(* Logix 5000 project; controller ARS14002_PLC vendor 1 type 14 code 218 rev 30.11; software revision 30.01; part 11 of 13 *)
(* tags used below, declared in another part *)
   AN_1000C : CM_AI_SCL;
   AN_1000C_SP : INT;
   AN_200A : CM_AI_SCL;
   AN_200A_SP : REAL;
   AT2_HIBON_DISCHARGE_TEMP_MAX : REAL;
   AT2_PLANT_ATOMIZING : BOOL;
   AT2_PLANT_ATOMIZING_ONS : BOOL;
   AT2_PLANT_COLLECTING : BOOL;
   AT2_PLANT_COLLECTION_TIME : TIMER;
   AT2_PLANT_GOOD_GAS_TIME : TIMER;   // AT2 total time with good gas and no collection stops
   AT2_PLANT_GOOD_H2O_TIME : TIMER;   // AT2 time with good dew point and no collection stop
   AT2_PLANT_GOOD_O2_TIME : TIMER;   // AT2 time with good O2 and no collection stop
   AT2_PLANT_H2O_MIN : REAL;   // AT2 Heat Minimum after burp
   AT2_PLANT_LIKELY_COLLECTING : BOOL;
   AT2_PLANT_LIKELY_COLLECTION_TIME : TIMER;
   AT2_PLANT_MAX_H2O : REAL;
   AT2_PLANT_MAX_O2 : REAL;
   AT2_PLANT_O2_MIN : REAL;   // AT2 Heat Minimum after burp
   AT3_HIBON_DISCHARGE_TEMP_MAX : REAL;
   AT3_PLANT_ATOMIZING : BOOL;
   AT3_PLANT_ATOMIZING_ONS : BOOL;
   AT3_PLANT_COLLECTING : BOOL;
   AT3_PLANT_COLLECTION_TIME : TIMER;
   AT3_PLANT_GOOD_GAS_TIME : TIMER;   // total time with good gas and no collection stops
   AT3_PLANT_GOOD_H2O_TIME : TIMER;   // time with good dew point and no collection stop
   AT3_PLANT_GOOD_O2_TIME : TIMER;   // time with good O2 and no collection stop
   AT3_PLANT_H2O_MIN : REAL;   // AT3 Plant Minimum after burp
   AT3_PLANT_LIKELY_COLLECTING : BOOL;
   AT3_PLANT_LIKELY_COLLECTION_TIME : TIMER;
   AT3_PLANT_MAX_H2O : REAL;
   AT3_PLANT_MAX_O2 : REAL;
   AT3_PLANT_O2_MIN : REAL;   // AT3 Plant Minimum after burp
   CALC_FT_1002_MONTH_RETURN : REAL;
   CALC_FT_1002_MONTH_TOTALIZER_RESET : BOOL;
   CALC_FT_1002_MONTH_TOTALIZER_START : BOOL;
   CALC_FT_1002_MONTH_TOTALIZER_STOP : BOOL;
   Calc_FT_1002_Return_Total : DINT[2100,13];
   Calc_Month : INT;
   CALC_NEXT_DAY_OSR_OB : BOOL;
   CALC_NEXT_DAY_OSR_SB : BOOL;
   CALC_NEXT_MONTH_OSR_OB : BOOL;
   CALC_NEXT_MONTH_OSR_SB : BOOL;
   Calc_TK_700_Fill_Lvl : REAL;
   Calc_TK_700_Fill_Start_Lvl : REAL;
   Calc_TK_700_Fill_Total : DINT[2100,13];
   Calc_TK_700_Month_Fill : REAL;
   Calc_TK_700_Month_Totalizer_Start : BOOL;
   Calc_TK_700_Month_Totalizer_Stop : BOOL;
   Calc_Year : INT;
   Collect_Stop_Dew_Pt : BOOL;
   Collect_Stop_O2 : BOOL;
   COLLECTION_ESTIMATE_SCALING_FACTOR : REAL;
   COLLECTION_LIKELY_PERCENTAGE : REAL;
   Cooldown_Complete_ONS_OB : BOOL;
   Cooldown_Complete_ONS_SB : BOOL;
   COOLDOWN_CYCLES_MIN : DINT[10];
   COOLDOWN_CYCLES_SEC : DINT[10];
   COOLDOWN_TIMER1 : TIMER;
   COOLDOWN_TIMER1_MIN : DINT;
   COOLDOWN_TIMER1_MS : DINT;
   COOLDOWN_TIMER1_SEC : DINT;
   CP_Run : BOOL;
   CP_Run_Atomize : BOOL;
   CP_Run_ONS_OB : BOOL;
   CP_Run_Standby : BOOL;
   CP_RUN_TIMESTAMP_DAY : DINT[10];
   CP_RUN_TIMESTAMP_HOUR : DINT[10];
   CP_RUN_TIMESTAMP_MIN : DINT[10];
   CP_RUN_TIMESTAMP_MONTH : DINT[10];
   CP_RUN_TIMESTAMP_SEC : DINT[10];
   CP_RUN_TIMESTAMP_YEAR : DINT[10];
   FCV_1002 : CM_AO_VLV;
   FCV_101A : CM_AO_VLV;
   FCV_101B : CM_AO_VLV;
   FCV_101C : CM_AO_VLV;
   FCV_102A : CM_AO_VLV;
   FCV_102B : CM_AO_VLV;
   FCV_102C : CM_AO_VLV;
   FCV_202 : CM_AO_VLV;
   FCV_202_COLLECTION_CERTAIN_SP : REAL;
   FCV_202_COLLECTION_LIKELY_SP : REAL;
   FCV_202_OPEN_DLA_TMR : TIMER;
   FCV_204 : CM_AO_VLV;
   FCV_207 : CM_AO_VLV;
   FIT_202_COLLECTION_FLOW : REAL;
   FT_1002 : CM_AI_SCL;
   FT_202 : CM_AI_SCL;
   FVR_800C_EN : BOOL;
   FVR_800D_EN : BOOL;
   HEAT_TIMER_AT2 : TIMER;
   HEAT_TIMER_AT3 : TIMER;
   HEAT_TIMER_PILOT : TIMER;
   P_800A_Cooldown_Complete : BOOL;
   P_800A_Start_Vent_TMR : TIMER;
   P_800B_Cooldown_Complete : BOOL;
   P_800B_Start_Vent_TMR : TIMER;
   P_800C_Cooldown_Complete : BOOL;
   P_800C_Start_Vent_TMR : TIMER;
   P_800D_Cooldown_Complete : BOOL;
   P_800D_Start_Vent_TMR : TIMER;
   PDT_701 : CM_AI_SCL_ALT;
   PIDE_1001 : PID_ENHANCED;
   PIDE_1002 : PID_ENHANCED;
   PIDE_1002_FLOW_SP : PID_ENHANCED;
   PIDE_1221 : PID_ENHANCED;
   PIDE_1251 : PID_ENHANCED;
   PIDE_603 : PID_ENHANCED;
   PIDE_605 : PID_ENHANCED;
   PIDE_753 : PID_ENHANCED;
   PIDE_754 : PID_ENHANCED;
   PIDE_755 : PID_ENHANCED;
   PIDE_800 : PID_ENHANCED;
   PILOT_PLANT_ATOMIZING : BOOL;
   PILOT_PLANT_ATOMIZING_ONS : BOOL;
   PILOT_PLANT_COLLECTING : BOOL;
   PILOT_PLANT_COLLECTION_PERCENT : REAL;
   PILOT_PLANT_COLLECTION_PERCENT_GOOD_GAS : REAL;
   PILOT_PLANT_COLLECTION_TIME : TIMER;
   PILOT_PLANT_GOOD_GAS_PERCENT : REAL;
   PILOT_PLANT_GOOD_GAS_TIME : TIMER;   // PILOT time with good gas and no collection stops
   PILOT_PLANT_GOOD_H2O_PERCENT : REAL;
   PILOT_PLANT_GOOD_H2O_TIME : TIMER;   // PILOT time with good dew point and no collection stop
   PILOT_PLANT_GOOD_O2_PERCENT : REAL;
   PILOT_PLANT_GOOD_O2_TIME : TIMER;   // PILOT time with good O2 and no collection stop
   PILOT_PLANT_H2O_MIN : REAL;   // Pilot Heat Minimum after burp
   PILOT_PLANT_LIKELY_COLLECTING : BOOL;
   PILOT_PLANT_LIKELY_COLLECTION_TIME : TIMER;
   PILOT_PLANT_MAX_H2O : REAL;
   PILOT_PLANT_MAX_O2 : REAL;
   PILOT_PLANT_O2_MIN : REAL;   // Pilot Heat Minimum after burp
   SV_1001F : CM_DO_GENERIC;
   SV_1002F : CM_DO_GENERIC;
   SV_1005X : CM_DO_GENERIC;
   SV_1221F : CM_DO_GENERIC;
   SV_1251F : CM_DO_GENERIC;
   SV_207F : CM_DO_GENERIC;
   SV_603F : CM_DO_GENERIC;
   SV_605F : CM_DO_GENERIC;
   SV_703X : CM_DO_GENERIC;
   SV_753F : CM_DO_GENERIC;
   SV_754F : CM_DO_GENERIC;
   SV_755F : CM_DO_GENERIC;
   TIME_TO_GOOD_GAS_AT2 : REAL;
   TIME_TO_GOOD_GAS_AT3 : REAL;
   TIME_TO_GOOD_GAS_PILOT : REAL;
   TimeStamp : DINT[7];
   VENT_COLLECTION_CERTAIN_SP : REAL;
   VENT_COLLECTION_LIKELY_SP : REAL;
   VFD_800A_EN : BOOL;
   VFD_800B_EN : BOOL;
   XV_1001 : CM_DO_VLV;
   XV_1123 : CM_DO_VLV;
   XV_1201 : CM_DO_VLV;
   XV_1202 : CM_DO_VLV;
   XV_1203 : CM_DO_VLV;
   ZT_1001 : CM_AI_SCL;
   ZT_207 : CM_AI_SCL;
(* MainProgram, continued *)

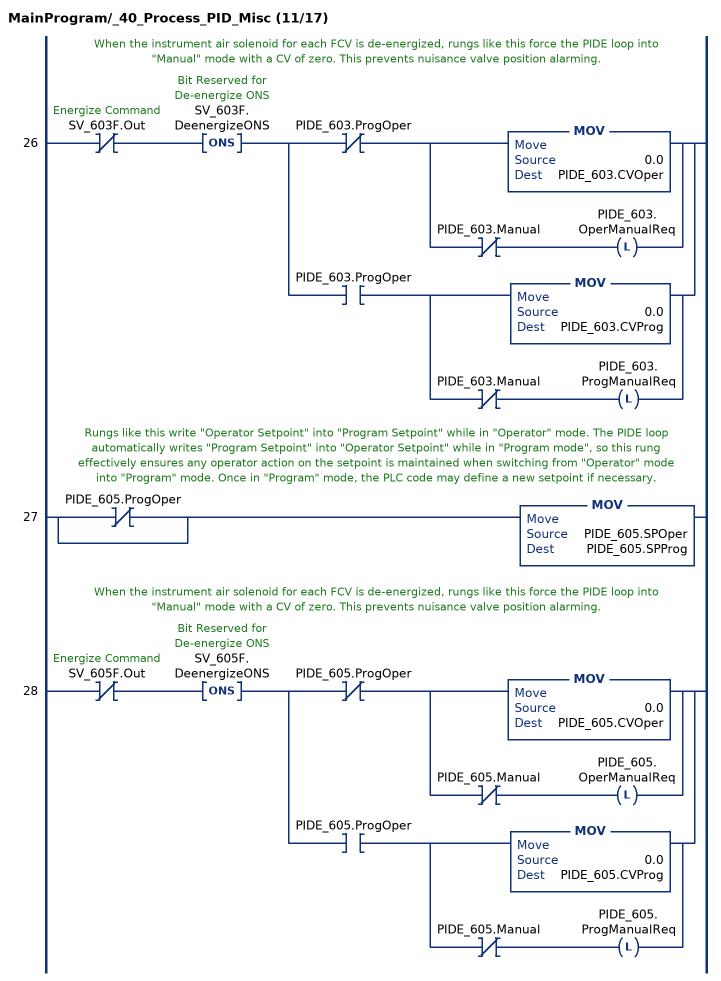
   [picture p222: MainProgram/_40_Process_PID_Misc rungs 26-28]
   // When the instrument air solenoid for each FCV is de-energized, rungs like this force the PIDE loop into "Manual" mode with a CV of zero. This prevents nuisance valve position alarming.
   26: XIO(SV_603F.Out)ONS(SV_603F.DeenergizeONS)[XIO(PIDE_603.ProgOper) [MOV(0.0,PIDE_603.CVOper) ,XIO(PIDE_603.Manual) OTL(PIDE_603.OperManualReq) ] ,XIC(PIDE_603.ProgOper) [MOV(0.0,PIDE_603.CVProg) ,XIO(PIDE_603.Manual) OTL(PIDE_603.ProgManualReq) ] ];
   // Rungs like this write "Operator Setpoint" into "Program Setpoint" while in "Operator" mode. The PIDE loop automatically writes "Program Setpoint" into "Operator Setpoint" while in "Program mode", so this rung effectively ensures any operator action on the setpoint is maintained when switching from "Operator" mode into "Program" mode. Once in "Program" mode, the PLC code may define a new setpoint if necessary.
   27: [XIO(PIDE_605.ProgOper) ,]MOV(PIDE_605.SPOper,PIDE_605.SPProg);
   // When the instrument air solenoid for each FCV is de-energized, rungs like this force the PIDE loop into "Manual" mode with a CV of zero. This prevents nuisance valve position alarming.
   28: XIO(SV_605F.Out)ONS(SV_605F.DeenergizeONS)[XIO(PIDE_605.ProgOper) [MOV(0.0,PIDE_605.CVOper) ,XIO(PIDE_605.Manual) OTL(PIDE_605.OperManualReq) ] ,XIC(PIDE_605.ProgOper) [MOV(0.0,PIDE_605.CVProg) ,XIO(PIDE_605.Manual) OTL(PIDE_605.ProgManualReq) ] ];
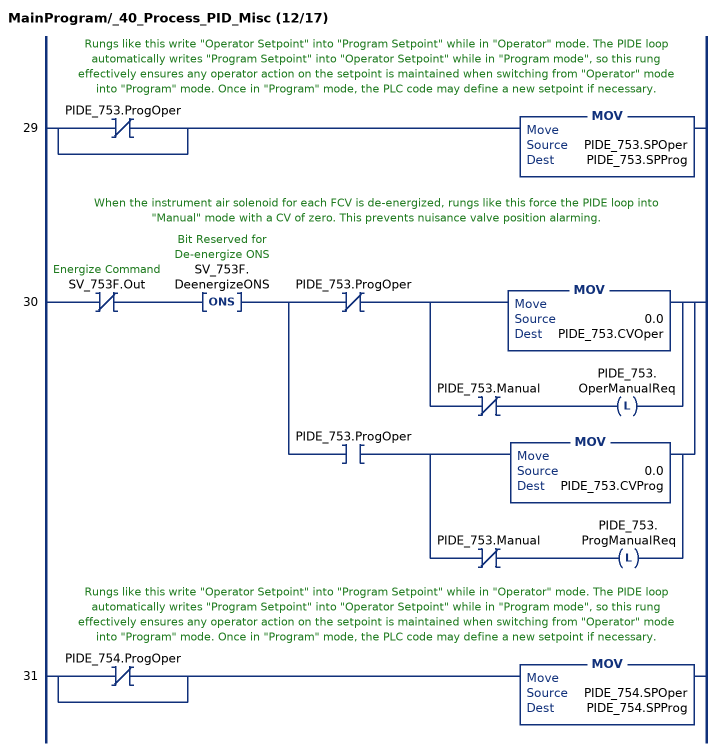
   // Rungs like this write "Operator Setpoint" into "Program Setpoint" while in "Operator" mode. The PIDE loop automatically writes "Program Setpoint" into "Operator Setpoint" while in "Program mode", so this rung effectively ensures any operator action on the setpoint is maintained when switching from "Operator" mode into "Program" mode. Once in "Program" mode, the PLC code may define a new setpoint if necessary.
   29: [XIO(PIDE_753.ProgOper) ,]MOV(PIDE_753.SPOper,PIDE_753.SPProg);
   // When the instrument air solenoid for each FCV is de-energized, rungs like this force the PIDE loop into "Manual" mode with a CV of zero. This prevents nuisance valve position alarming.
   30: XIO(SV_753F.Out)ONS(SV_753F.DeenergizeONS)[XIO(PIDE_753.ProgOper) [MOV(0.0,PIDE_753.CVOper) ,XIO(PIDE_753.Manual) OTL(PIDE_753.OperManualReq) ] ,XIC(PIDE_753.ProgOper) [MOV(0.0,PIDE_753.CVProg) ,XIO(PIDE_753.Manual) OTL(PIDE_753.ProgManualReq) ] ];
   // Rungs like this write "Operator Setpoint" into "Program Setpoint" while in "Operator" mode. The PIDE loop automatically writes "Program Setpoint" into "Operator Setpoint" while in "Program mode", so this rung effectively ensures any operator action on the setpoint is maintained when switching from "Operator" mode into "Program" mode. Once in "Program" mode, the PLC code may define a new setpoint if necessary.
   31: [XIO(PIDE_754.ProgOper) ,]MOV(PIDE_754.SPOper,PIDE_754.SPProg);
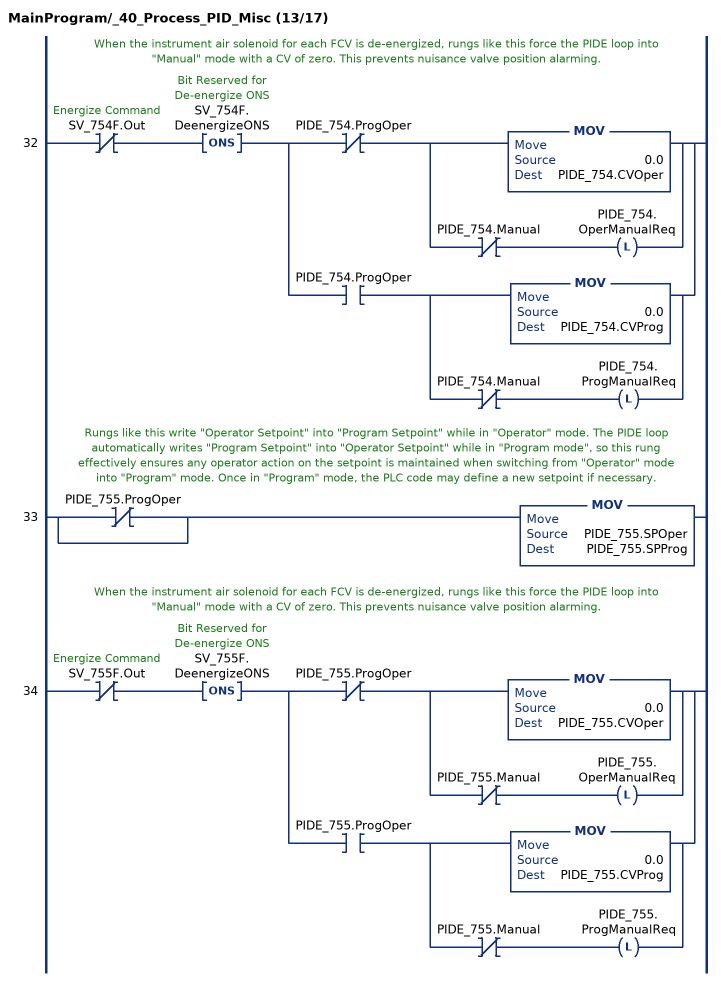
   // When the instrument air solenoid for each FCV is de-energized, rungs like this force the PIDE loop into "Manual" mode with a CV of zero. This prevents nuisance valve position alarming.
   32: XIO(SV_754F.Out)ONS(SV_754F.DeenergizeONS)[XIO(PIDE_754.ProgOper) [MOV(0.0,PIDE_754.CVOper) ,XIO(PIDE_754.Manual) OTL(PIDE_754.OperManualReq) ] ,XIC(PIDE_754.ProgOper) [MOV(0.0,PIDE_754.CVProg) ,XIO(PIDE_754.Manual) OTL(PIDE_754.ProgManualReq) ] ];
   // Rungs like this write "Operator Setpoint" into "Program Setpoint" while in "Operator" mode. The PIDE loop automatically writes "Program Setpoint" into "Operator Setpoint" while in "Program mode", so this rung effectively ensures any operator action on the setpoint is maintained when switching from "Operator" mode into "Program" mode. Once in "Program" mode, the PLC code may define a new setpoint if necessary.
   33: [XIO(PIDE_755.ProgOper) ,]MOV(PIDE_755.SPOper,PIDE_755.SPProg);
   // When the instrument air solenoid for each FCV is de-energized, rungs like this force the PIDE loop into "Manual" mode with a CV of zero. This prevents nuisance valve position alarming.
   34: XIO(SV_755F.Out)ONS(SV_755F.DeenergizeONS)[XIO(PIDE_755.ProgOper) [MOV(0.0,PIDE_755.CVOper) ,XIO(PIDE_755.Manual) OTL(PIDE_755.OperManualReq) ] ,XIC(PIDE_755.ProgOper) [MOV(0.0,PIDE_755.CVProg) ,XIO(PIDE_755.Manual) OTL(PIDE_755.ProgManualReq) ] ];
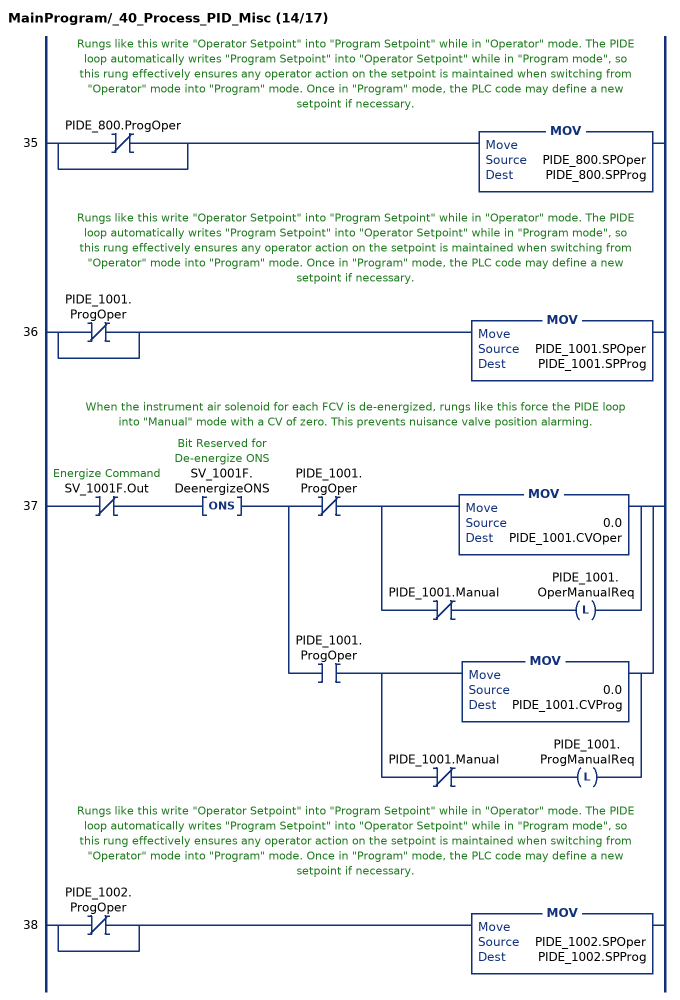
   // Rungs like this write "Operator Setpoint" into "Program Setpoint" while in "Operator" mode. The PIDE loop automatically writes "Program Setpoint" into "Operator Setpoint" while in "Program mode", so this rung effectively ensures any operator action on the setpoint is maintained when switching from "Operator" mode into "Program" mode. Once in "Program" mode, the PLC code may define a new setpoint if necessary.
   35: [XIO(PIDE_800.ProgOper) ,]MOV(PIDE_800.SPOper,PIDE_800.SPProg);
   // Rungs like this write "Operator Setpoint" into "Program Setpoint" while in "Operator" mode. The PIDE loop automatically writes "Program Setpoint" into "Operator Setpoint" while in "Program mode", so this rung effectively ensures any operator action on the setpoint is maintained when switching from "Operator" mode into "Program" mode. Once in "Program" mode, the PLC code may define a new setpoint if necessary.
   36: [XIO(PIDE_1001.ProgOper) ,]MOV(PIDE_1001.SPOper,PIDE_1001.SPProg);
   // When the instrument air solenoid for each FCV is de-energized, rungs like this force the PIDE loop into "Manual" mode with a CV of zero. This prevents nuisance valve position alarming.
   37: XIO(SV_1001F.Out)ONS(SV_1001F.DeenergizeONS)[XIO(PIDE_1001.ProgOper) [MOV(0.0,PIDE_1001.CVOper) ,XIO(PIDE_1001.Manual) OTL(PIDE_1001.OperManualReq) ] ,XIC(PIDE_1001.ProgOper) [MOV(0.0,PIDE_1001.CVProg) ,XIO(PIDE_1001.Manual) OTL(PIDE_1001.ProgManualReq) ] ];
   // Rungs like this write "Operator Setpoint" into "Program Setpoint" while in "Operator" mode. The PIDE loop automatically writes "Program Setpoint" into "Operator Setpoint" while in "Program mode", so this rung effectively ensures any operator action on the setpoint is maintained when switching from "Operator" mode into "Program" mode. Once in "Program" mode, the PLC code may define a new setpoint if necessary.
   38: [XIO(PIDE_1002.ProgOper) ,]MOV(PIDE_1002.SPOper,PIDE_1002.SPProg);
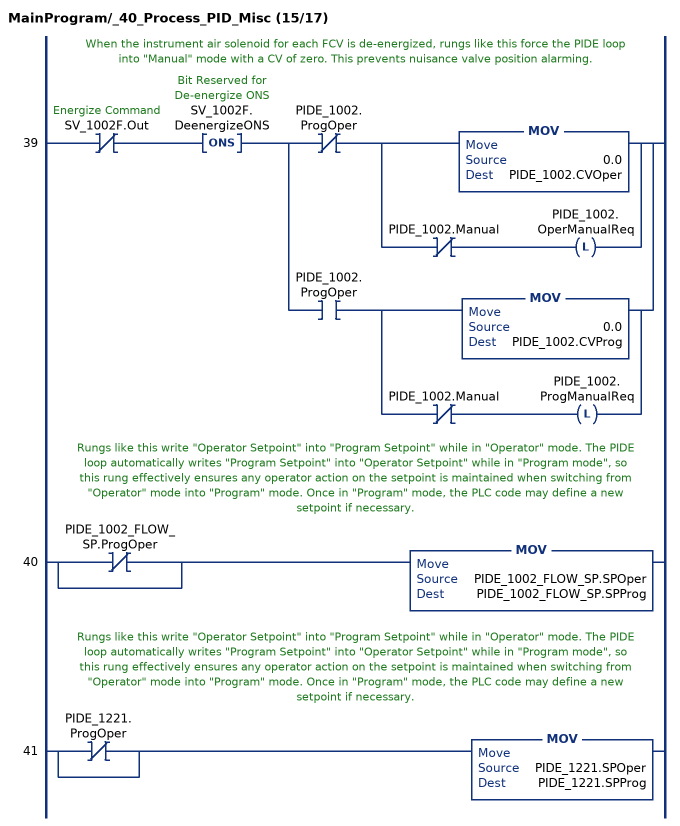
   // When the instrument air solenoid for each FCV is de-energized, rungs like this force the PIDE loop into "Manual" mode with a CV of zero. This prevents nuisance valve position alarming.
   39: XIO(SV_1002F.Out)ONS(SV_1002F.DeenergizeONS)[XIO(PIDE_1002.ProgOper) [MOV(0.0,PIDE_1002.CVOper) ,XIO(PIDE_1002.Manual) OTL(PIDE_1002.OperManualReq) ] ,XIC(PIDE_1002.ProgOper) [MOV(0.0,PIDE_1002.CVProg) ,XIO(PIDE_1002.Manual) OTL(PIDE_1002.ProgManualReq) ] ];
   // Rungs like this write "Operator Setpoint" into "Program Setpoint" while in "Operator" mode. The PIDE loop automatically writes "Program Setpoint" into "Operator Setpoint" while in "Program mode", so this rung effectively ensures any operator action on the setpoint is maintained when switching from "Operator" mode into "Program" mode. Once in "Program" mode, the PLC code may define a new setpoint if necessary.
   40: [XIO(PIDE_1002_FLOW_SP.ProgOper) ,]MOV(PIDE_1002_FLOW_SP.SPOper,PIDE_1002_FLOW_SP.SPProg);
   // Rungs like this write "Operator Setpoint" into "Program Setpoint" while in "Operator" mode. The PIDE loop automatically writes "Program Setpoint" into "Operator Setpoint" while in "Program mode", so this rung effectively ensures any operator action on the setpoint is maintained when switching from "Operator" mode into "Program" mode. Once in "Program" mode, the PLC code may define a new setpoint if necessary.
   41: [XIO(PIDE_1221.ProgOper) ,]MOV(PIDE_1221.SPOper,PIDE_1221.SPProg);
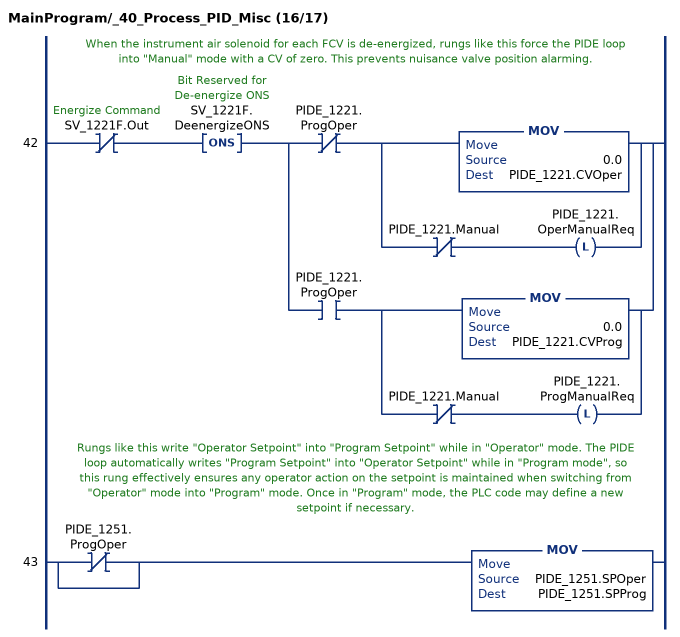
   // When the instrument air solenoid for each FCV is de-energized, rungs like this force the PIDE loop into "Manual" mode with a CV of zero. This prevents nuisance valve position alarming.
   42: XIO(SV_1221F.Out)ONS(SV_1221F.DeenergizeONS)[XIO(PIDE_1221.ProgOper) [MOV(0.0,PIDE_1221.CVOper) ,XIO(PIDE_1221.Manual) OTL(PIDE_1221.OperManualReq) ] ,XIC(PIDE_1221.ProgOper) [MOV(0.0,PIDE_1221.CVProg) ,XIO(PIDE_1221.Manual) OTL(PIDE_1221.ProgManualReq) ] ];
   // Rungs like this write "Operator Setpoint" into "Program Setpoint" while in "Operator" mode. The PIDE loop automatically writes "Program Setpoint" into "Operator Setpoint" while in "Program mode", so this rung effectively ensures any operator action on the setpoint is maintained when switching from "Operator" mode into "Program" mode. Once in "Program" mode, the PLC code may define a new setpoint if necessary.
   43: [XIO(PIDE_1251.ProgOper) ,]MOV(PIDE_1251.SPOper,PIDE_1251.SPProg);
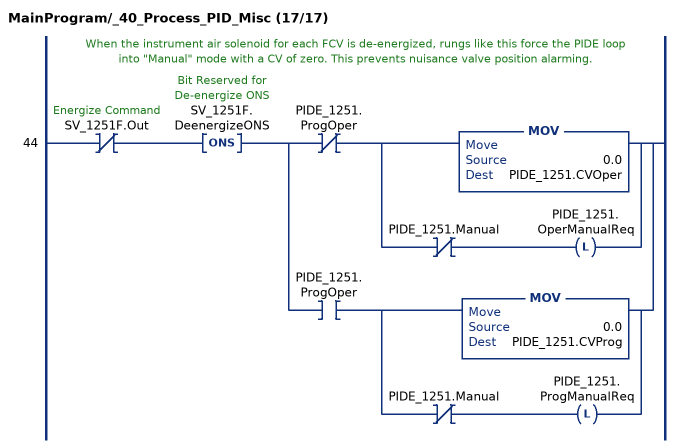
   // When the instrument air solenoid for each FCV is de-energized, rungs like this force the PIDE loop into "Manual" mode with a CV of zero. This prevents nuisance valve position alarming.
   44: XIO(SV_1251F.Out)ONS(SV_1251F.DeenergizeONS)[XIO(PIDE_1251.ProgOper) [MOV(0.0,PIDE_1251.CVOper) ,XIO(PIDE_1251.Manual) OTL(PIDE_1251.OperManualReq) ] ,XIC(PIDE_1251.ProgOper) [MOV(0.0,PIDE_1251.CVProg) ,XIO(PIDE_1251.Manual) OTL(PIDE_1251.ProgManualReq) ] ];
END_ROUTINE

ROUTINE _41_Data_Table_Logging   (* ladder *)
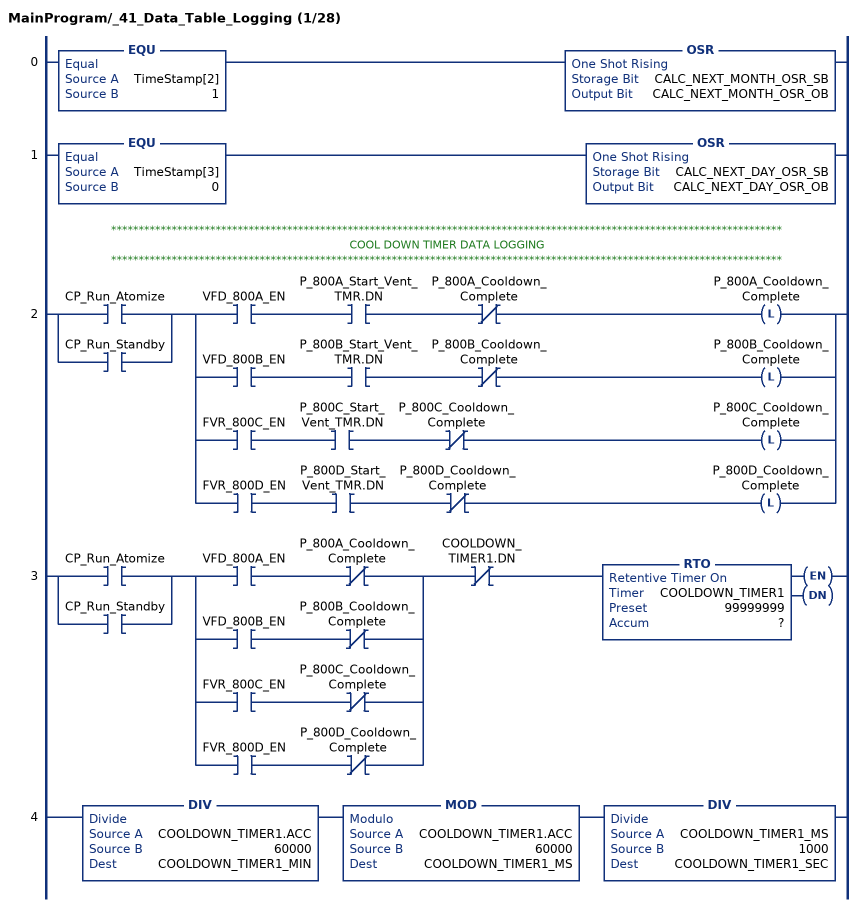
   0: EQU(TimeStamp[2],1)OSR(CALC_NEXT_MONTH_OSR_SB,CALC_NEXT_MONTH_OSR_OB);
   1: EQU(TimeStamp[3],0)OSR(CALC_NEXT_DAY_OSR_SB,CALC_NEXT_DAY_OSR_OB);
   // **************************************************************************************************************************
   // COOL DOWN TIMER DATA LOGGING
   // **************************************************************************************************************************
   2: [XIC(CP_Run_Atomize) ,XIC(CP_Run_Standby) ][XIC(VFD_800A_EN) XIC(P_800A_Start_Vent_TMR.DN) XIO(P_800A_Cooldown_Complete) OTL(P_800A_Cooldown_Complete) ,XIC(VFD_800B_EN) XIC(P_800B_Start_Vent_TMR.DN) XIO(P_800B_Cooldown_Complete) OTL(P_800B_Cooldown_Complete) ,XIC(FVR_800C_EN) XIC(P_800C_Start_Vent_TMR.DN) XIO(P_800C_Cooldown_Complete) OTL(P_800C_Cooldown_Complete) ,XIC(FVR_800D_EN) XIC(P_800D_Start_Vent_TMR.DN) XIO(P_800D_Cooldown_Complete) OTL(P_800D_Cooldown_Complete) ];
   3: [XIC(CP_Run_Atomize) ,XIC(CP_Run_Standby) ][XIC(VFD_800A_EN) XIO(P_800A_Cooldown_Complete) ,XIC(VFD_800B_EN) XIO(P_800B_Cooldown_Complete) ,XIC(FVR_800C_EN) XIO(P_800C_Cooldown_Complete) ,XIC(FVR_800D_EN) XIO(P_800D_Cooldown_Complete) ]XIO(COOLDOWN_TIMER1.DN)RTO(COOLDOWN_TIMER1,?,?);
   4: DIV(COOLDOWN_TIMER1.ACC,60000,COOLDOWN_TIMER1_MIN)MOD(COOLDOWN_TIMER1.ACC,60000,COOLDOWN_TIMER1_MS)DIV(COOLDOWN_TIMER1_MS,1000,COOLDOWN_TIMER1_SEC);
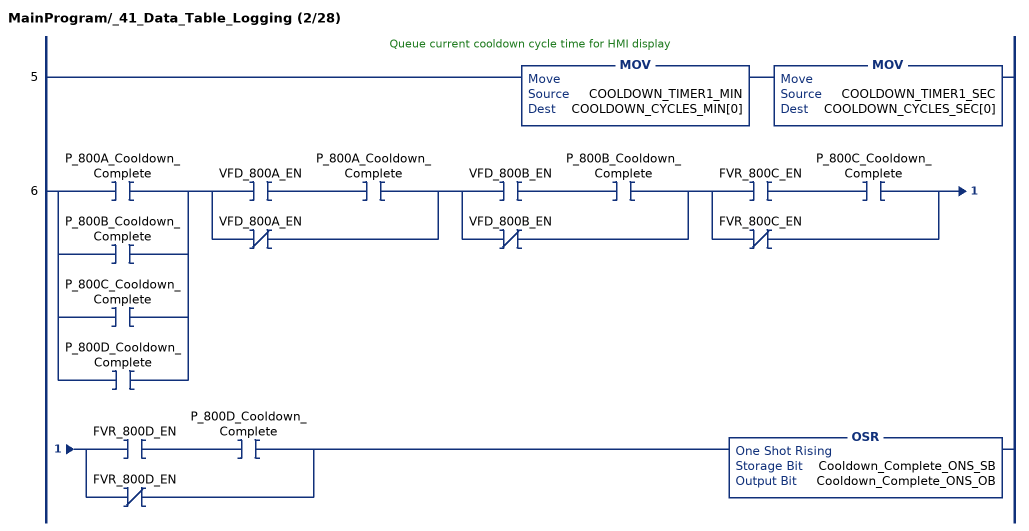
   // Queue current cooldown cycle time for HMI display
   5: MOV(COOLDOWN_TIMER1_MIN,COOLDOWN_CYCLES_MIN[0])MOV(COOLDOWN_TIMER1_SEC,COOLDOWN_CYCLES_SEC[0]);
   6: [XIC(P_800A_Cooldown_Complete) ,XIC(P_800B_Cooldown_Complete) ,XIC(P_800C_Cooldown_Complete) ,XIC(P_800D_Cooldown_Complete) ][XIC(VFD_800A_EN) XIC(P_800A_Cooldown_Complete) ,XIO(VFD_800A_EN) ][XIC(VFD_800B_EN) XIC(P_800B_Cooldown_Complete) ,XIO(VFD_800B_EN) ][XIC(FVR_800C_EN) XIC(P_800C_Cooldown_Complete) ,XIO(FVR_800C_EN) ][XIC(FVR_800D_EN) XIC(P_800D_Cooldown_Complete) ,XIO(FVR_800D_EN) ]OSR(Cooldown_Complete_ONS_SB,Cooldown_Complete_ONS_OB);
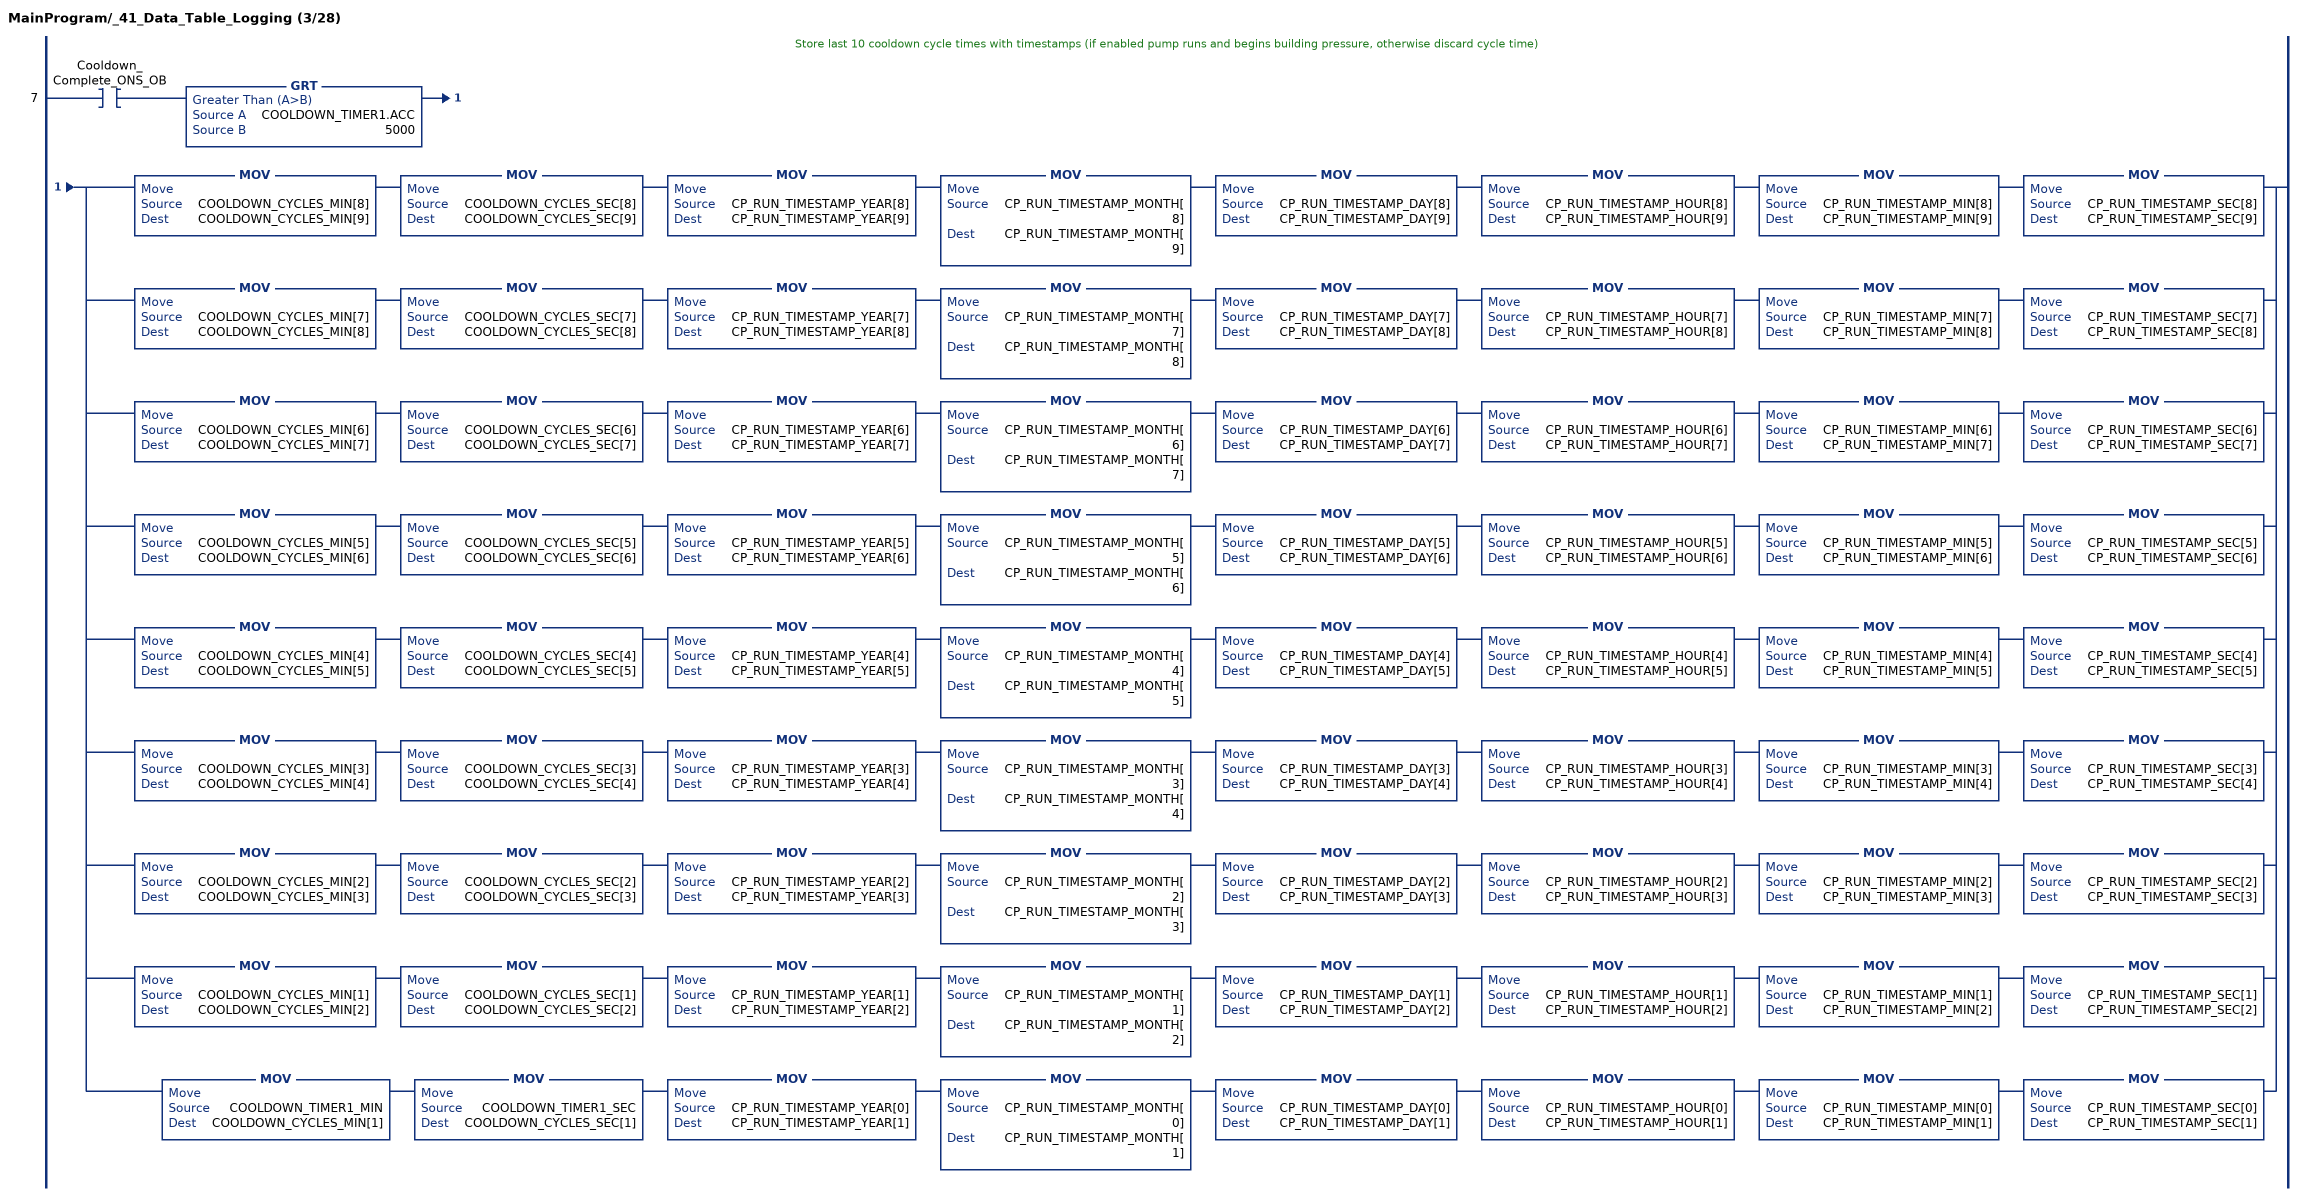
   // Store last 10 cooldown cycle times with timestamps (if enabled pump runs and begins building pressure, otherwise discard cycle time)
   7: XIC(Cooldown_Complete_ONS_OB)GRT(COOLDOWN_TIMER1.ACC,5000)[MOV(COOLDOWN_CYCLES_MIN[8],COOLDOWN_CYCLES_MIN[9]) MOV(COOLDOWN_CYCLES_SEC[8],COOLDOWN_CYCLES_SEC[9]) MOV(CP_RUN_TIMESTAMP_YEAR[8],CP_RUN_TIMESTAMP_YEAR[9]) MOV(CP_RUN_TIMESTAMP_MONTH[8],CP_RUN_TIMESTAMP_MONTH[9]) MOV(CP_RUN_TIMESTAMP_DAY[8],CP_RUN_TIMESTAMP_DAY[9]) MOV(CP_RUN_TIMESTAMP_HOUR[8],CP_RUN_TIMESTAMP_HOUR[9]) MOV(CP_RUN_TIMESTAMP_MIN[8],CP_RUN_TIMESTAMP_MIN[9]) MOV(CP_RUN_TIMESTAMP_SEC[8],CP_RUN_TIMESTAMP_SEC[9]) ,MOV(COOLDOWN_CYCLES_MIN[7],COOLDOWN_CYCLES_MIN[8]) MOV(COOLDOWN_CYCLES_SEC[7],COOLDOWN_CYCLES_SEC[8]) MOV(CP_RUN_TIMESTAMP_YEAR[7],CP_RUN_TIMESTAMP_YEAR[8]) MOV(CP_RUN_TIMESTAMP_MONTH[7],CP_RUN_TIMESTAMP_MONTH[8]) MOV(CP_RUN_TIMESTAMP_DAY[7],CP_RUN_TIMESTAMP_DAY[8]) MOV(CP_RUN_TIMESTAMP_HOUR[7],CP_RUN_TIMESTAMP_HOUR[8]) MOV(CP_RUN_TIMESTAMP_MIN[7],CP_RUN_TIMESTAMP_MIN[8]) MOV(CP_RUN_TIMESTAMP_SEC[7],CP_RUN_TIMESTAMP_SEC[8]) ,MOV(COOLDOWN_CYCLES_MIN[6],COOLDOWN_CYCLES_MIN[7]) MOV(COOLDOWN_CYCLES_SEC[6],COOLDOWN_CYCLES_SEC[7]) MOV(CP_RUN_TIMESTAMP_YEAR[6],CP_RUN_TIMESTAMP_YEAR[7]) MOV(CP_RUN_TIMESTAMP_MONTH[6],CP_RUN_TIMESTAMP_MONTH[7]) MOV(CP_RUN_TIMESTAMP_DAY[6],CP_RUN_TIMESTAMP_DAY[7]) MOV(CP_RUN_TIMESTAMP_HOUR[6],CP_RUN_TIMESTAMP_HOUR[7]) MOV(CP_RUN_TIMESTAMP_MIN[6],CP_RUN_TIMESTAMP_MIN[7]) MOV(CP_RUN_TIMESTAMP_SEC[6],CP_RUN_TIMESTAMP_SEC[7]) ,MOV(COOLDOWN_CYCLES_MIN[5],COOLDOWN_CYCLES_MIN[6]) MOV(COOLDOWN_CYCLES_SEC[5],COOLDOWN_CYCLES_SEC[6]) MOV(CP_RUN_TIMESTAMP_YEAR[5],CP_RUN_TIMESTAMP_YEAR[6]) MOV(CP_RUN_TIMESTAMP_MONTH[5],CP_RUN_TIMESTAMP_MONTH[6]) MOV(CP_RUN_TIMESTAMP_DAY[5],CP_RUN_TIMESTAMP_DAY[6]) MOV(CP_RUN_TIMESTAMP_HOUR[5],CP_RUN_TIMESTAMP_HOUR[6]) MOV(CP_RUN_TIMESTAMP_MIN[5],CP_RUN_TIMESTAMP_MIN[6]) MOV(CP_RUN_TIMESTAMP_SEC[5],CP_RUN_TIMESTAMP_SEC[6]) ,MOV(COOLDOWN_CYCLES_MIN[4],COOLDOWN_CYCLES_MIN[5]) MOV(COOLDOWN_CYCLES_SEC[4],COOLDOWN_CYCLES_SEC[5]) MOV(CP_RUN_TIMESTAMP_YEAR[4],CP_RUN_TIMESTAMP_YEAR[5]) MOV(CP_RUN_TIMESTAMP_MONTH[4],CP_RUN_TIMESTAMP_MONTH[5]) MOV(CP_RUN_TIMESTAMP_DAY[4],CP_RUN_TIMESTAMP_DAY[5]) MOV(CP_RUN_TIMESTAMP_HOUR[4],CP_RUN_TIMESTAMP_HOUR[5]) MOV(CP_RUN_TIMESTAMP_MIN[4],CP_RUN_TIMESTAMP_MIN[5]) MOV(CP_RUN_TIMESTAMP_SEC[4],CP_RUN_TIMESTAMP_SEC[5]) ,MOV(COOLDOWN_CYCLES_MIN[3],COOLDOWN_CYCLES_MIN[4]) MOV(COOLDOWN_CYCLES_SEC[3],COOLDOWN_CYCLES_SEC[4]) MOV(CP_RUN_TIMESTAMP_YEAR[3],CP_RUN_TIMESTAMP_YEAR[4]) MOV(CP_RUN_TIMESTAMP_MONTH[3],CP_RUN_TIMESTAMP_MONTH[4]) MOV(CP_RUN_TIMESTAMP_DAY[3],CP_RUN_TIMESTAMP_DAY[4]) MOV(CP_RUN_TIMESTAMP_HOUR[3],CP_RUN_TIMESTAMP_HOUR[4]) MOV(CP_RUN_TIMESTAMP_MIN[3],CP_RUN_TIMESTAMP_MIN[4]) MOV(CP_RUN_TIMESTAMP_SEC[3],CP_RUN_TIMESTAMP_SEC[4]) ,MOV(COOLDOWN_CYCLES_MIN[2],COOLDOWN_CYCLES_MIN[3]) MOV(COOLDOWN_CYCLES_SEC[2],COOLDOWN_CYCLES_SEC[3]) MOV(CP_RUN_TIMESTAMP_YEAR[2],CP_RUN_TIMESTAMP_YEAR[3]) MOV(CP_RUN_TIMESTAMP_MONTH[2],CP_RUN_TIMESTAMP_MONTH[3]) MOV(CP_RUN_TIMESTAMP_DAY[2],CP_RUN_TIMESTAMP_DAY[3]) MOV(CP_RUN_TIMESTAMP_HOUR[2],CP_RUN_TIMESTAMP_HOUR[3]) MOV(CP_RUN_TIMESTAMP_MIN[2],CP_RUN_TIMESTAMP_MIN[3]) MOV(CP_RUN_TIMESTAMP_SEC[2],CP_RUN_TIMESTAMP_SEC[3]) ,MOV(COOLDOWN_CYCLES_MIN[1],COOLDOWN_CYCLES_MIN[2]) MOV(COOLDOWN_CYCLES_SEC[1],COOLDOWN_CYCLES_SEC[2]) MOV(CP_RUN_TIMESTAMP_YEAR[1],CP_RUN_TIMESTAMP_YEAR[2]) MOV(CP_RUN_TIMESTAMP_MONTH[1],CP_RUN_TIMESTAMP_MONTH[2]) MOV(CP_RUN_TIMESTAMP_DAY[1],CP_RUN_TIMESTAMP_DAY[2]) MOV(CP_RUN_TIMESTAMP_HOUR[1],CP_RUN_TIMESTAMP_HOUR[2]) MOV(CP_RUN_TIMESTAMP_MIN[1],CP_RUN_TIMESTAMP_MIN[2]) MOV(CP_RUN_TIMESTAMP_SEC[1],CP_RUN_TIMESTAMP_SEC[2]) ,MOV(COOLDOWN_TIMER1_MIN,COOLDOWN_CYCLES_MIN[1]) MOV(COOLDOWN_TIMER1_SEC,COOLDOWN_CYCLES_SEC[1]) MOV(CP_RUN_TIMESTAMP_YEAR[0],CP_RUN_TIMESTAMP_YEAR[1]) MOV(CP_RUN_TIMESTAMP_MONTH[0],CP_RUN_TIMESTAMP_MONTH[1]) MOV(CP_RUN_TIMESTAMP_DAY[0],CP_RUN_TIMESTAMP_DAY[1]) MOV(CP_RUN_TIMESTAMP_HOUR[0],CP_RUN_TIMESTAMP_HOUR[1]) MOV(CP_RUN_TIMESTAMP_MIN[0],CP_RUN_TIMESTAMP_MIN[1]) MOV(CP_RUN_TIMESTAMP_SEC[0],CP_RUN_TIMESTAMP_SEC[1]) ];
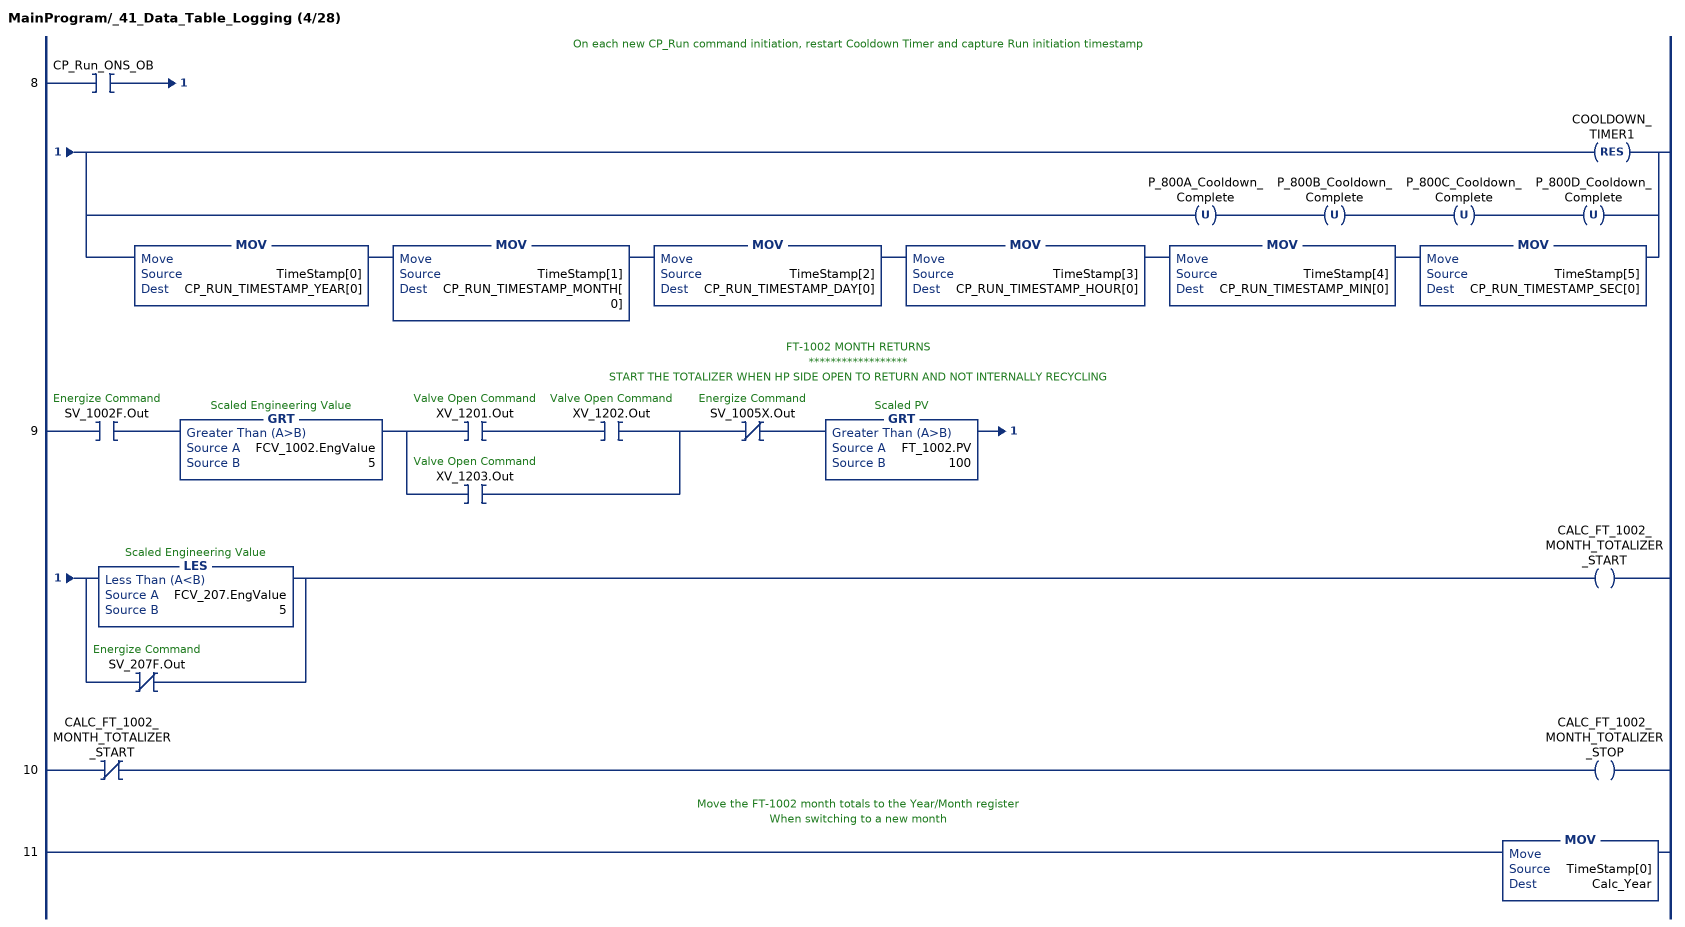
   // On each new CP_Run command initiation, restart Cooldown Timer and capture Run initiation timestamp
   8: XIC(CP_Run_ONS_OB)[[RES(COOLDOWN_TIMER1) ,OTU(P_800A_Cooldown_Complete) OTU(P_800B_Cooldown_Complete) OTU(P_800C_Cooldown_Complete) OTU(P_800D_Cooldown_Complete) ] ,MOV(TimeStamp[0],CP_RUN_TIMESTAMP_YEAR[0]) MOV(TimeStamp[1],CP_RUN_TIMESTAMP_MONTH[0]) MOV(TimeStamp[2],CP_RUN_TIMESTAMP_DAY[0]) MOV(TimeStamp[3],CP_RUN_TIMESTAMP_HOUR[0]) MOV(TimeStamp[4],CP_RUN_TIMESTAMP_MIN[0]) MOV(TimeStamp[5],CP_RUN_TIMESTAMP_SEC[0]) ];
   // FT-1002 MONTH RETURNS
   // ******************
   // START THE TOTALIZER WHEN HP SIDE OPEN TO RETURN AND NOT INTERNALLY RECYCLING
   9: XIC(SV_1002F.Out)GRT(FCV_1002.EngValue,5)[XIC(XV_1201.Out) XIC(XV_1202.Out) ,XIC(XV_1203.Out) ]XIO(SV_1005X.Out)GRT(FT_1002.PV,100)[LES(FCV_207.EngValue,5) ,XIO(SV_207F.Out) ]OTE(CALC_FT_1002_MONTH_TOTALIZER_START);
   10: XIO(CALC_FT_1002_MONTH_TOTALIZER_START)OTE(CALC_FT_1002_MONTH_TOTALIZER_STOP);
   // Move the FT-1002 month totals to the Year/Month register
   // When switching to a new month
   11: MOV(TimeStamp[0],Calc_Year);
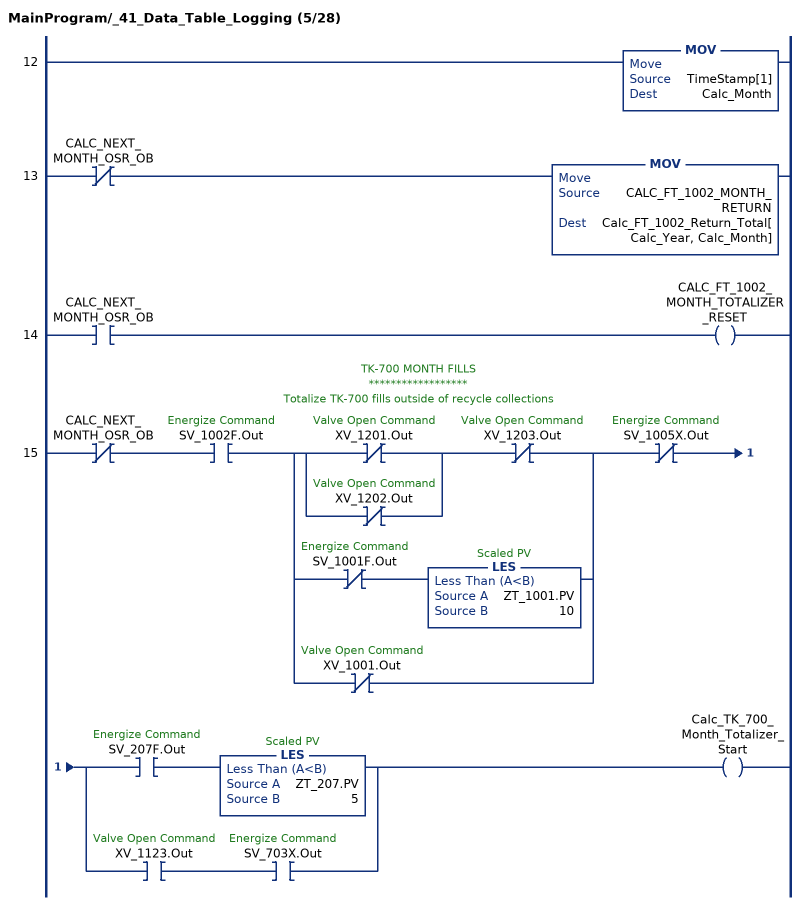
   12: MOV(TimeStamp[1],Calc_Month);
   13: XIO(CALC_NEXT_MONTH_OSR_OB)MOV(CALC_FT_1002_MONTH_RETURN,Calc_FT_1002_Return_Total[Calc_Year, Calc_Month]);
   14: XIC(CALC_NEXT_MONTH_OSR_OB)OTE(CALC_FT_1002_MONTH_TOTALIZER_RESET);
   // TK-700 MONTH FILLS
   // ******************
   // Totalize TK-700 fills outside of recycle collections
   15: XIO(CALC_NEXT_MONTH_OSR_OB)XIC(SV_1002F.Out)[[XIO(XV_1201.Out) ,XIO(XV_1202.Out) ] XIO(XV_1203.Out) ,XIO(SV_1001F.Out) LES(ZT_1001.PV,10) ,XIO(XV_1001.Out) ]XIO(SV_1005X.Out)[XIC(SV_207F.Out) LES(ZT_207.PV,5) ,XIC(XV_1123.Out) XIC(SV_703X.Out) ]OTE(Calc_TK_700_Month_Totalizer_Start);
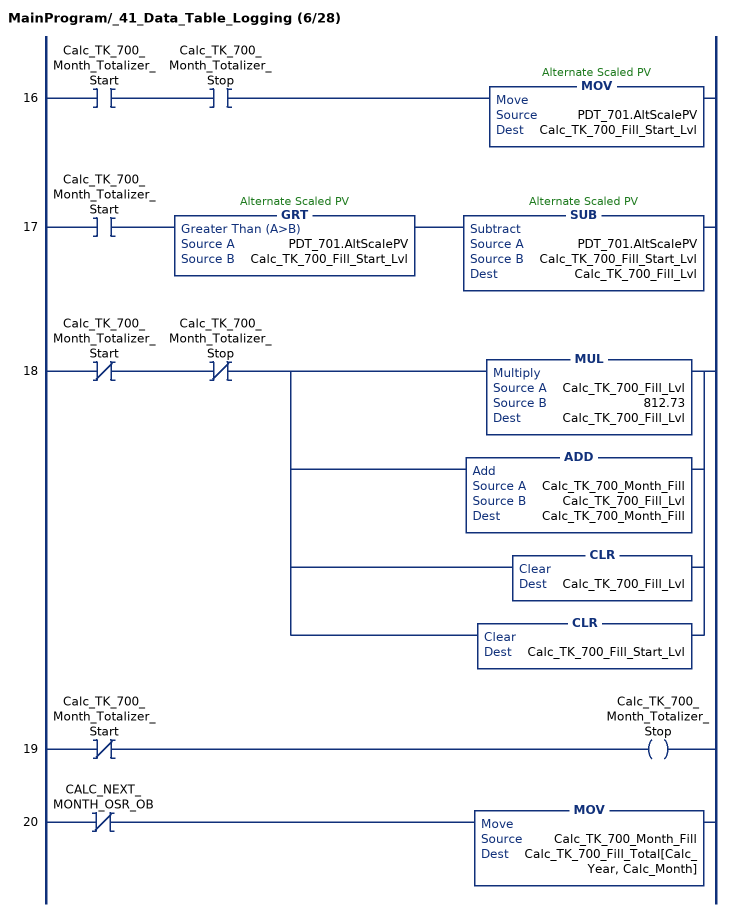
   16: XIC(Calc_TK_700_Month_Totalizer_Start)XIC(Calc_TK_700_Month_Totalizer_Stop)MOV(PDT_701.AltScalePV,Calc_TK_700_Fill_Start_Lvl);
   17: XIC(Calc_TK_700_Month_Totalizer_Start)GRT(PDT_701.AltScalePV,Calc_TK_700_Fill_Start_Lvl)SUB(PDT_701.AltScalePV,Calc_TK_700_Fill_Start_Lvl,Calc_TK_700_Fill_Lvl);
   18: XIO(Calc_TK_700_Month_Totalizer_Start)XIO(Calc_TK_700_Month_Totalizer_Stop)[MUL(Calc_TK_700_Fill_Lvl,812.73,Calc_TK_700_Fill_Lvl) ,ADD(Calc_TK_700_Month_Fill,Calc_TK_700_Fill_Lvl,Calc_TK_700_Month_Fill) ,CLR(Calc_TK_700_Fill_Lvl) ,CLR(Calc_TK_700_Fill_Start_Lvl) ];
   19: XIO(Calc_TK_700_Month_Totalizer_Start)OTE(Calc_TK_700_Month_Totalizer_Stop);
   20: XIO(CALC_NEXT_MONTH_OSR_OB)MOV(Calc_TK_700_Month_Fill,Calc_TK_700_Fill_Total[Calc_Year, Calc_Month]);
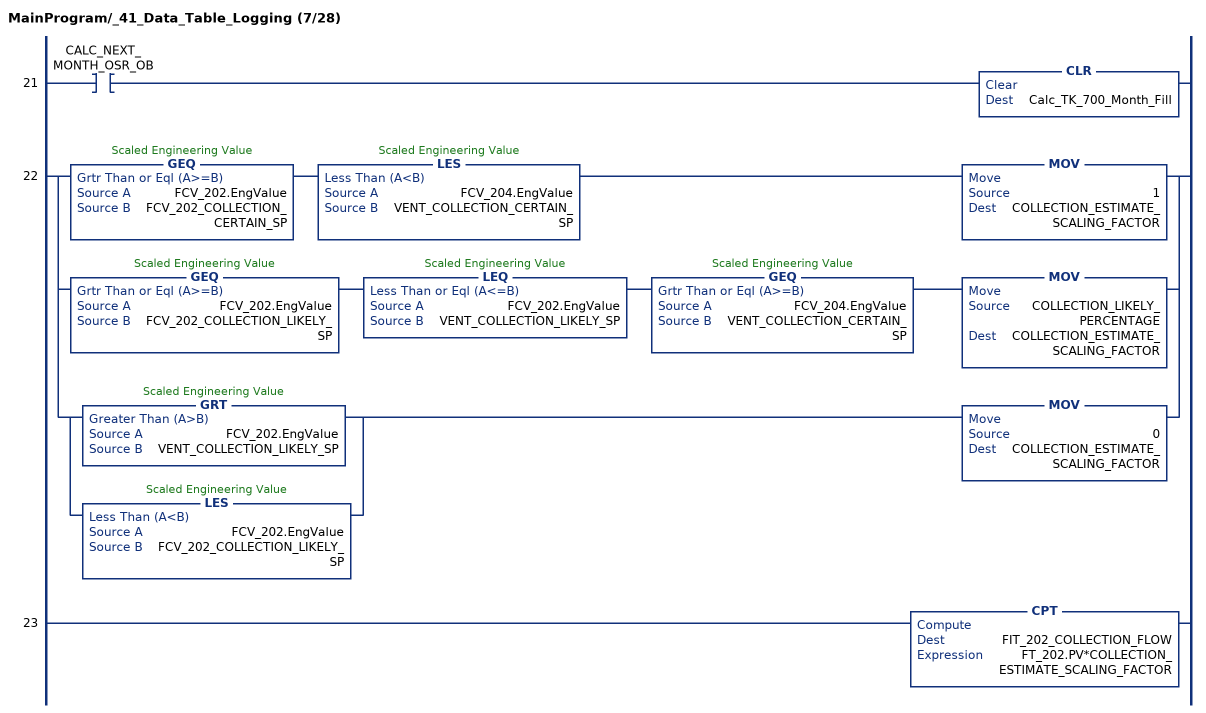
   21: XIC(CALC_NEXT_MONTH_OSR_OB)CLR(Calc_TK_700_Month_Fill);
   22: [GEQ(FCV_202.EngValue,FCV_202_COLLECTION_CERTAIN_SP) LES(FCV_204.EngValue,VENT_COLLECTION_CERTAIN_SP) MOV(1,COLLECTION_ESTIMATE_SCALING_FACTOR) ,GEQ(FCV_202.EngValue,FCV_202_COLLECTION_LIKELY_SP) LEQ(FCV_202.EngValue,VENT_COLLECTION_LIKELY_SP) GEQ(FCV_204.EngValue,VENT_COLLECTION_CERTAIN_SP) MOV(COLLECTION_LIKELY_PERCENTAGE,COLLECTION_ESTIMATE_SCALING_FACTOR) ,[GRT(FCV_202.EngValue,VENT_COLLECTION_LIKELY_SP) ,LES(FCV_202.EngValue,FCV_202_COLLECTION_LIKELY_SP) ] MOV(0,COLLECTION_ESTIMATE_SCALING_FACTOR) ];
   23: CPT(FIT_202_COLLECTION_FLOW,FT_202.PV*COLLECTION_ESTIMATE_SCALING_FACTOR);
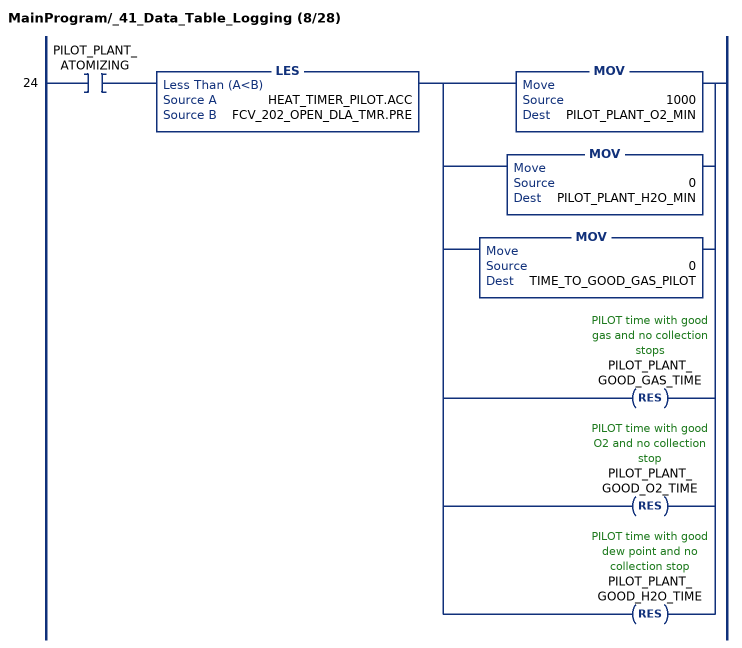
   24: XIC(PILOT_PLANT_ATOMIZING)LES(HEAT_TIMER_PILOT.ACC,FCV_202_OPEN_DLA_TMR.PRE)[MOV(1000,PILOT_PLANT_O2_MIN) ,MOV(0,PILOT_PLANT_H2O_MIN) ,MOV(0,TIME_TO_GOOD_GAS_PILOT) ,RES(PILOT_PLANT_GOOD_GAS_TIME) ,RES(PILOT_PLANT_GOOD_O2_TIME) ,RES(PILOT_PLANT_GOOD_H2O_TIME) ];
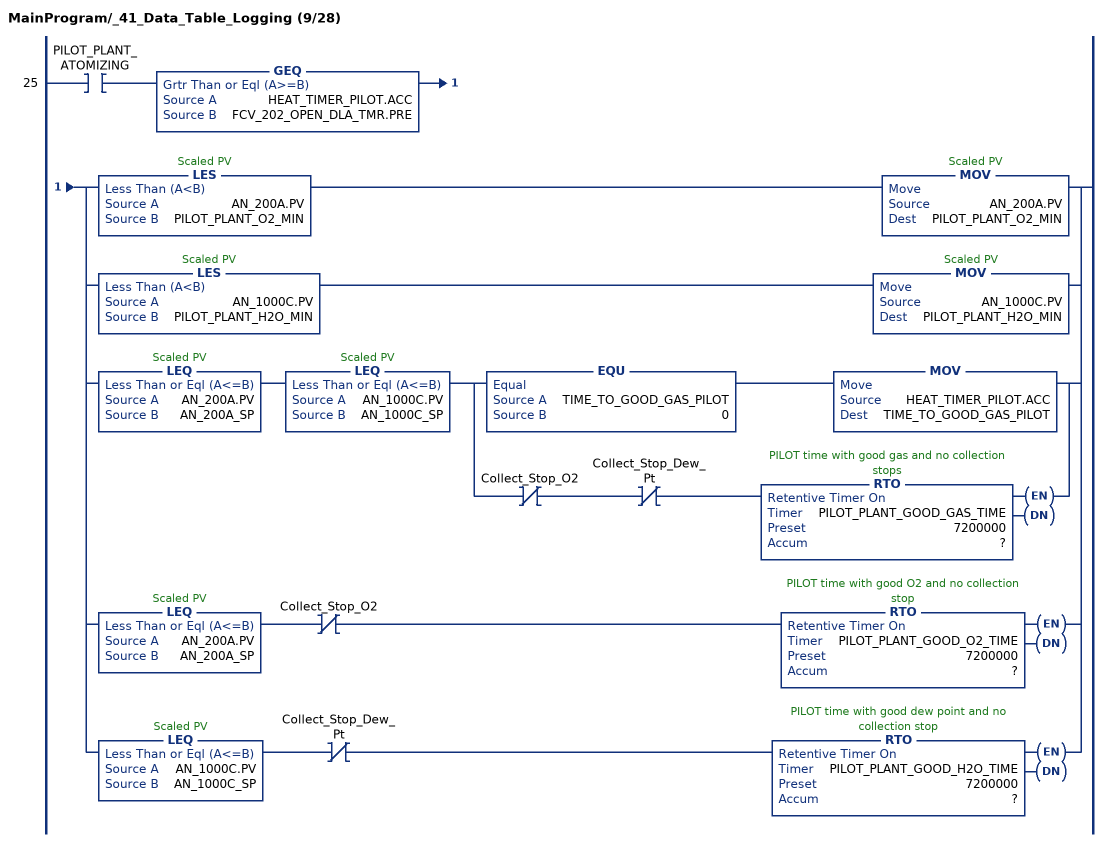
   25: XIC(PILOT_PLANT_ATOMIZING)GEQ(HEAT_TIMER_PILOT.ACC,FCV_202_OPEN_DLA_TMR.PRE)[LES(AN_200A.PV,PILOT_PLANT_O2_MIN) MOV(AN_200A.PV,PILOT_PLANT_O2_MIN) ,LES(AN_1000C.PV,PILOT_PLANT_H2O_MIN) MOV(AN_1000C.PV,PILOT_PLANT_H2O_MIN) ,LEQ(AN_200A.PV,AN_200A_SP) LEQ(AN_1000C.PV,AN_1000C_SP) [EQU(TIME_TO_GOOD_GAS_PILOT,0) MOV(HEAT_TIMER_PILOT.ACC,TIME_TO_GOOD_GAS_PILOT) ,XIO(Collect_Stop_O2) XIO(Collect_Stop_Dew_Pt) RTO(PILOT_PLANT_GOOD_GAS_TIME,?,?) ] ,LEQ(AN_200A.PV,AN_200A_SP) XIO(Collect_Stop_O2) RTO(PILOT_PLANT_GOOD_O2_TIME,?,?) ,LEQ(AN_1000C.PV,AN_1000C_SP) XIO(Collect_Stop_Dew_Pt) RTO(PILOT_PLANT_GOOD_H2O_TIME,?,?) ];
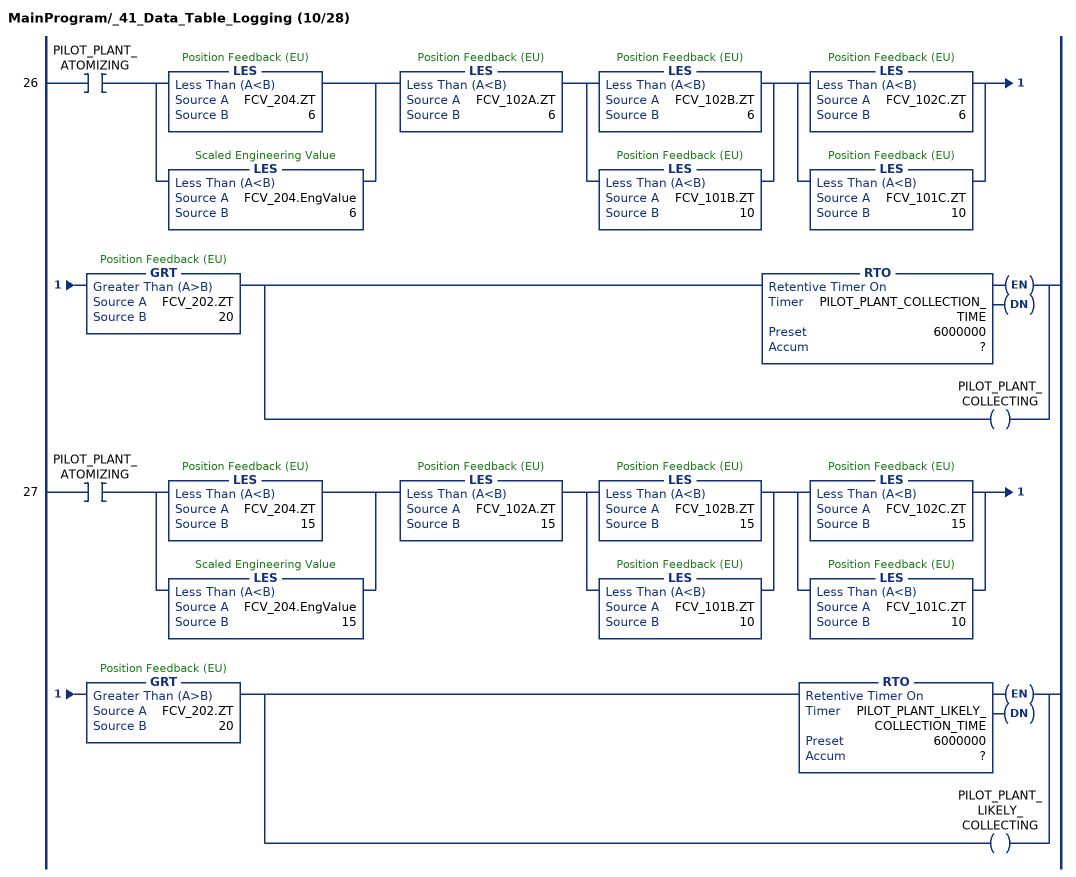
   26: XIC(PILOT_PLANT_ATOMIZING)[LES(FCV_204.ZT,6) ,LES(FCV_204.EngValue,6) ]LES(FCV_102A.ZT,6)[LES(FCV_102B.ZT,6) ,LES(FCV_101B.ZT,10) ][LES(FCV_102C.ZT,6) ,LES(FCV_101C.ZT,10) ]GRT(FCV_202.ZT,20)[RTO(PILOT_PLANT_COLLECTION_TIME,?,?) ,OTE(PILOT_PLANT_COLLECTING) ];
   27: XIC(PILOT_PLANT_ATOMIZING)[LES(FCV_204.ZT,15) ,LES(FCV_204.EngValue,15) ]LES(FCV_102A.ZT,15)[LES(FCV_102B.ZT,15) ,LES(FCV_101B.ZT,10) ][LES(FCV_102C.ZT,15) ,LES(FCV_101C.ZT,10) ]GRT(FCV_202.ZT,20)[RTO(PILOT_PLANT_LIKELY_COLLECTION_TIME,?,?) ,OTE(PILOT_PLANT_LIKELY_COLLECTING) ];
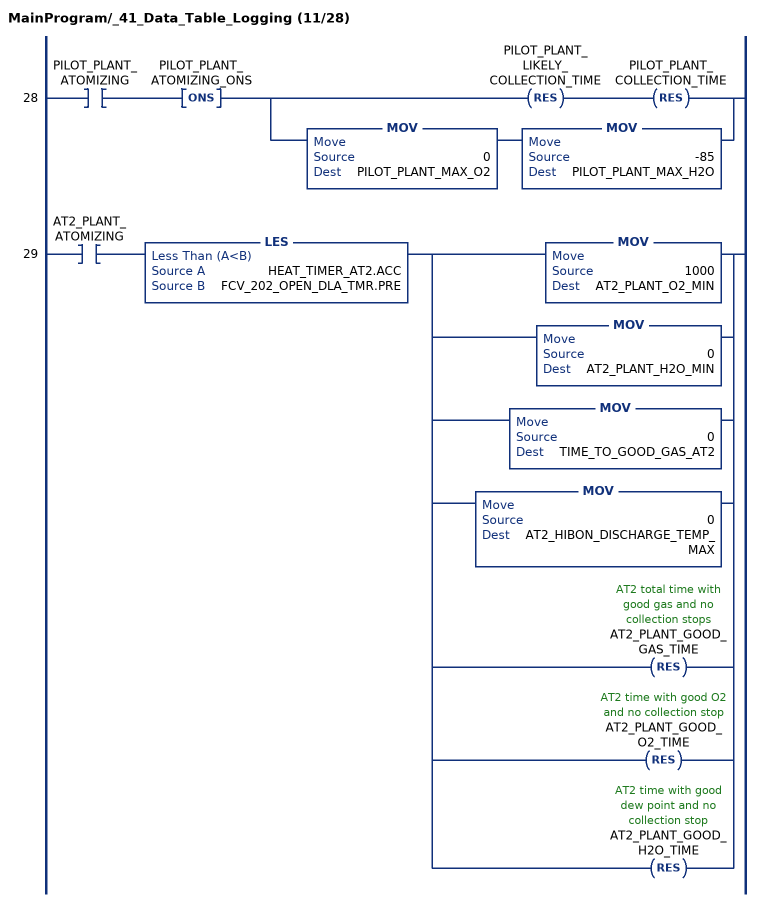
   28: XIC(PILOT_PLANT_ATOMIZING)ONS(PILOT_PLANT_ATOMIZING_ONS)[RES(PILOT_PLANT_LIKELY_COLLECTION_TIME) RES(PILOT_PLANT_COLLECTION_TIME) ,MOV(0,PILOT_PLANT_MAX_O2) MOV(-85,PILOT_PLANT_MAX_H2O) ];
   29: XIC(AT2_PLANT_ATOMIZING)LES(HEAT_TIMER_AT2.ACC,FCV_202_OPEN_DLA_TMR.PRE)[MOV(1000,AT2_PLANT_O2_MIN) ,MOV(0,AT2_PLANT_H2O_MIN) ,MOV(0,TIME_TO_GOOD_GAS_AT2) ,MOV(0,AT2_HIBON_DISCHARGE_TEMP_MAX) ,RES(AT2_PLANT_GOOD_GAS_TIME) ,RES(AT2_PLANT_GOOD_O2_TIME) ,RES(AT2_PLANT_GOOD_H2O_TIME) ];
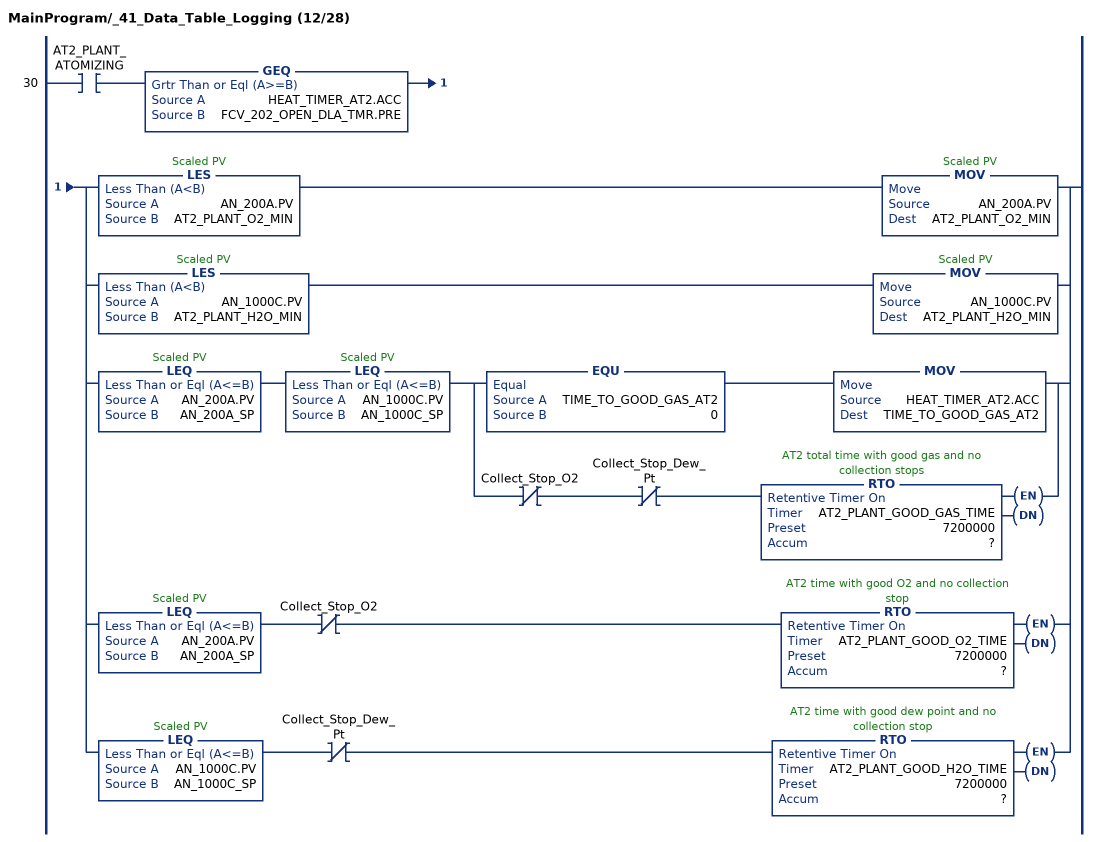
   30: XIC(AT2_PLANT_ATOMIZING)GEQ(HEAT_TIMER_AT2.ACC,FCV_202_OPEN_DLA_TMR.PRE)[LES(AN_200A.PV,AT2_PLANT_O2_MIN) MOV(AN_200A.PV,AT2_PLANT_O2_MIN) ,LES(AN_1000C.PV,AT2_PLANT_H2O_MIN) MOV(AN_1000C.PV,AT2_PLANT_H2O_MIN) ,LEQ(AN_200A.PV,AN_200A_SP) LEQ(AN_1000C.PV,AN_1000C_SP) [EQU(TIME_TO_GOOD_GAS_AT2,0) MOV(HEAT_TIMER_AT2.ACC,TIME_TO_GOOD_GAS_AT2) ,XIO(Collect_Stop_O2) XIO(Collect_Stop_Dew_Pt) RTO(AT2_PLANT_GOOD_GAS_TIME,?,?) ] ,LEQ(AN_200A.PV,AN_200A_SP) XIO(Collect_Stop_O2) RTO(AT2_PLANT_GOOD_O2_TIME,?,?) ,LEQ(AN_1000C.PV,AN_1000C_SP) XIO(Collect_Stop_Dew_Pt) RTO(AT2_PLANT_GOOD_H2O_TIME,?,?) ];
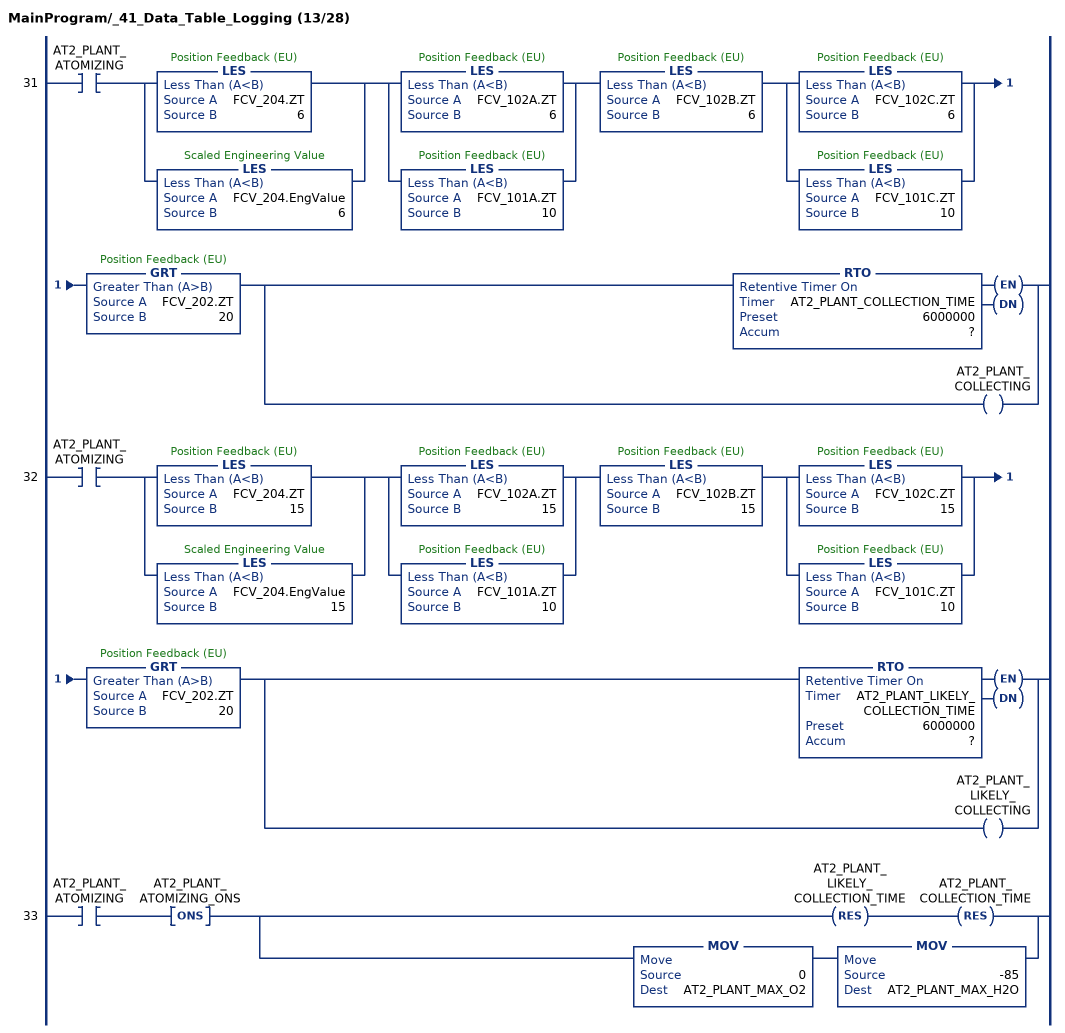
   31: XIC(AT2_PLANT_ATOMIZING)[LES(FCV_204.ZT,6) ,LES(FCV_204.EngValue,6) ][LES(FCV_102A.ZT,6) ,LES(FCV_101A.ZT,10) ]LES(FCV_102B.ZT,6)[LES(FCV_102C.ZT,6) ,LES(FCV_101C.ZT,10) ]GRT(FCV_202.ZT,20)[RTO(AT2_PLANT_COLLECTION_TIME,?,?) ,OTE(AT2_PLANT_COLLECTING) ];
   32: XIC(AT2_PLANT_ATOMIZING)[LES(FCV_204.ZT,15) ,LES(FCV_204.EngValue,15) ][LES(FCV_102A.ZT,15) ,LES(FCV_101A.ZT,10) ]LES(FCV_102B.ZT,15)[LES(FCV_102C.ZT,15) ,LES(FCV_101C.ZT,10) ]GRT(FCV_202.ZT,20)[RTO(AT2_PLANT_LIKELY_COLLECTION_TIME,?,?) ,OTE(AT2_PLANT_LIKELY_COLLECTING) ];
   33: XIC(AT2_PLANT_ATOMIZING)ONS(AT2_PLANT_ATOMIZING_ONS)[RES(AT2_PLANT_LIKELY_COLLECTION_TIME) RES(AT2_PLANT_COLLECTION_TIME) ,MOV(0,AT2_PLANT_MAX_O2) MOV(-85,AT2_PLANT_MAX_H2O) ];
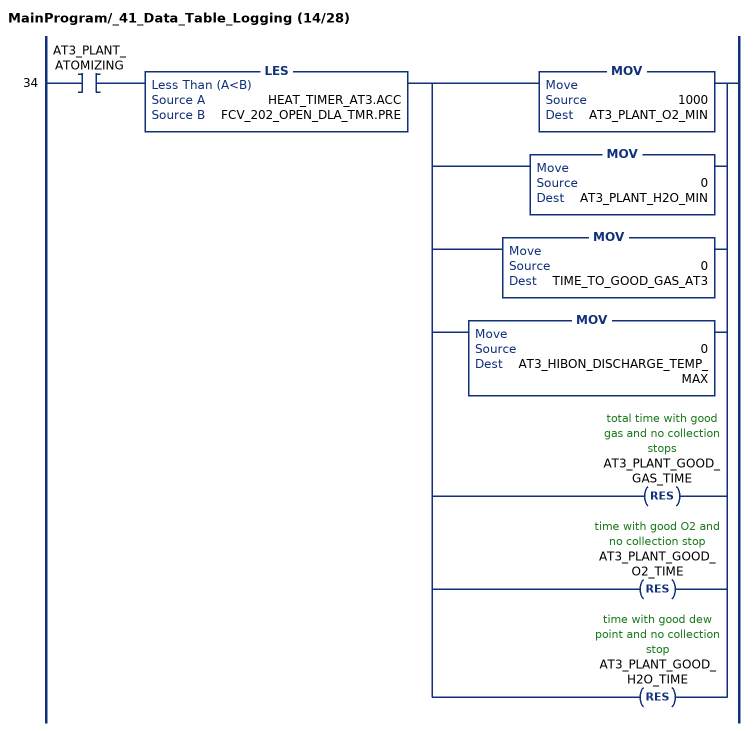
   34: XIC(AT3_PLANT_ATOMIZING)LES(HEAT_TIMER_AT3.ACC,FCV_202_OPEN_DLA_TMR.PRE)[MOV(1000,AT3_PLANT_O2_MIN) ,MOV(0,AT3_PLANT_H2O_MIN) ,MOV(0,TIME_TO_GOOD_GAS_AT3) ,MOV(0,AT3_HIBON_DISCHARGE_TEMP_MAX) ,RES(AT3_PLANT_GOOD_GAS_TIME) ,RES(AT3_PLANT_GOOD_O2_TIME) ,RES(AT3_PLANT_GOOD_H2O_TIME) ];
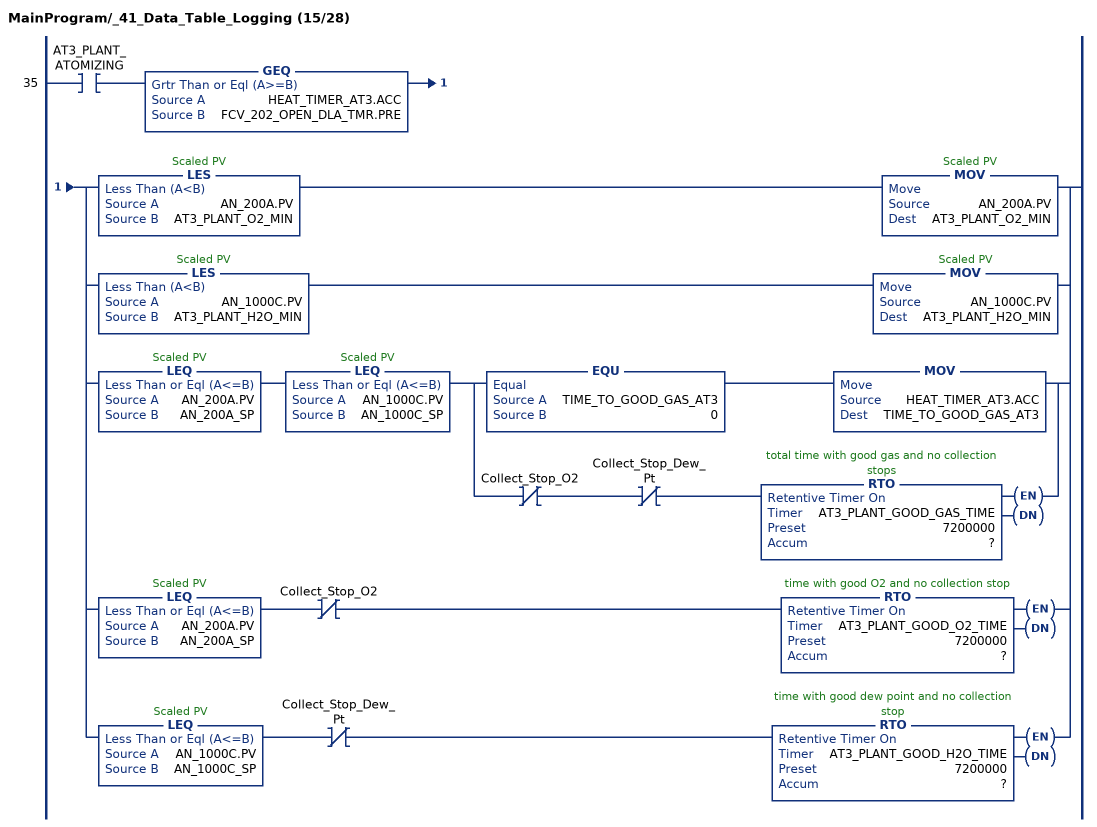
   35: XIC(AT3_PLANT_ATOMIZING)GEQ(HEAT_TIMER_AT3.ACC,FCV_202_OPEN_DLA_TMR.PRE)[LES(AN_200A.PV,AT3_PLANT_O2_MIN) MOV(AN_200A.PV,AT3_PLANT_O2_MIN) ,LES(AN_1000C.PV,AT3_PLANT_H2O_MIN) MOV(AN_1000C.PV,AT3_PLANT_H2O_MIN) ,LEQ(AN_200A.PV,AN_200A_SP) LEQ(AN_1000C.PV,AN_1000C_SP) [EQU(TIME_TO_GOOD_GAS_AT3,0) MOV(HEAT_TIMER_AT3.ACC,TIME_TO_GOOD_GAS_AT3) ,XIO(Collect_Stop_O2) XIO(Collect_Stop_Dew_Pt) RTO(AT3_PLANT_GOOD_GAS_TIME,?,?) ] ,LEQ(AN_200A.PV,AN_200A_SP) XIO(Collect_Stop_O2) RTO(AT3_PLANT_GOOD_O2_TIME,?,?) ,LEQ(AN_1000C.PV,AN_1000C_SP) XIO(Collect_Stop_Dew_Pt) RTO(AT3_PLANT_GOOD_H2O_TIME,?,?) ];
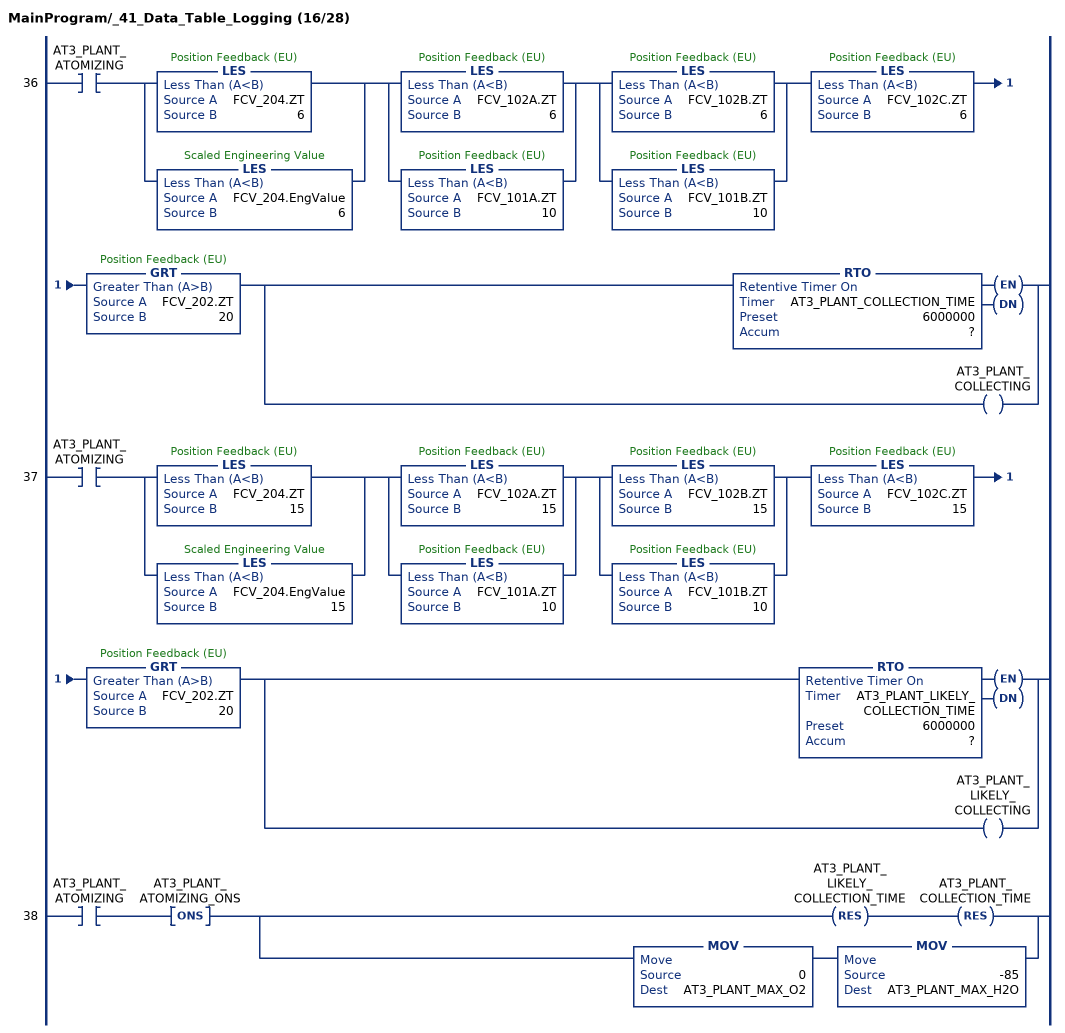
   36: XIC(AT3_PLANT_ATOMIZING)[LES(FCV_204.ZT,6) ,LES(FCV_204.EngValue,6) ][LES(FCV_102A.ZT,6) ,LES(FCV_101A.ZT,10) ][LES(FCV_102B.ZT,6) ,LES(FCV_101B.ZT,10) ]LES(FCV_102C.ZT,6)GRT(FCV_202.ZT,20)[RTO(AT3_PLANT_COLLECTION_TIME,?,?) ,OTE(AT3_PLANT_COLLECTING) ];
   37: XIC(AT3_PLANT_ATOMIZING)[LES(FCV_204.ZT,15) ,LES(FCV_204.EngValue,15) ][LES(FCV_102A.ZT,15) ,LES(FCV_101A.ZT,10) ][LES(FCV_102B.ZT,15) ,LES(FCV_101B.ZT,10) ]LES(FCV_102C.ZT,15)GRT(FCV_202.ZT,20)[RTO(AT3_PLANT_LIKELY_COLLECTION_TIME,?,?) ,OTE(AT3_PLANT_LIKELY_COLLECTING) ];
   38: XIC(AT3_PLANT_ATOMIZING)ONS(AT3_PLANT_ATOMIZING_ONS)[RES(AT3_PLANT_LIKELY_COLLECTION_TIME) RES(AT3_PLANT_COLLECTION_TIME) ,MOV(0,AT3_PLANT_MAX_O2) MOV(-85,AT3_PLANT_MAX_H2O) ];
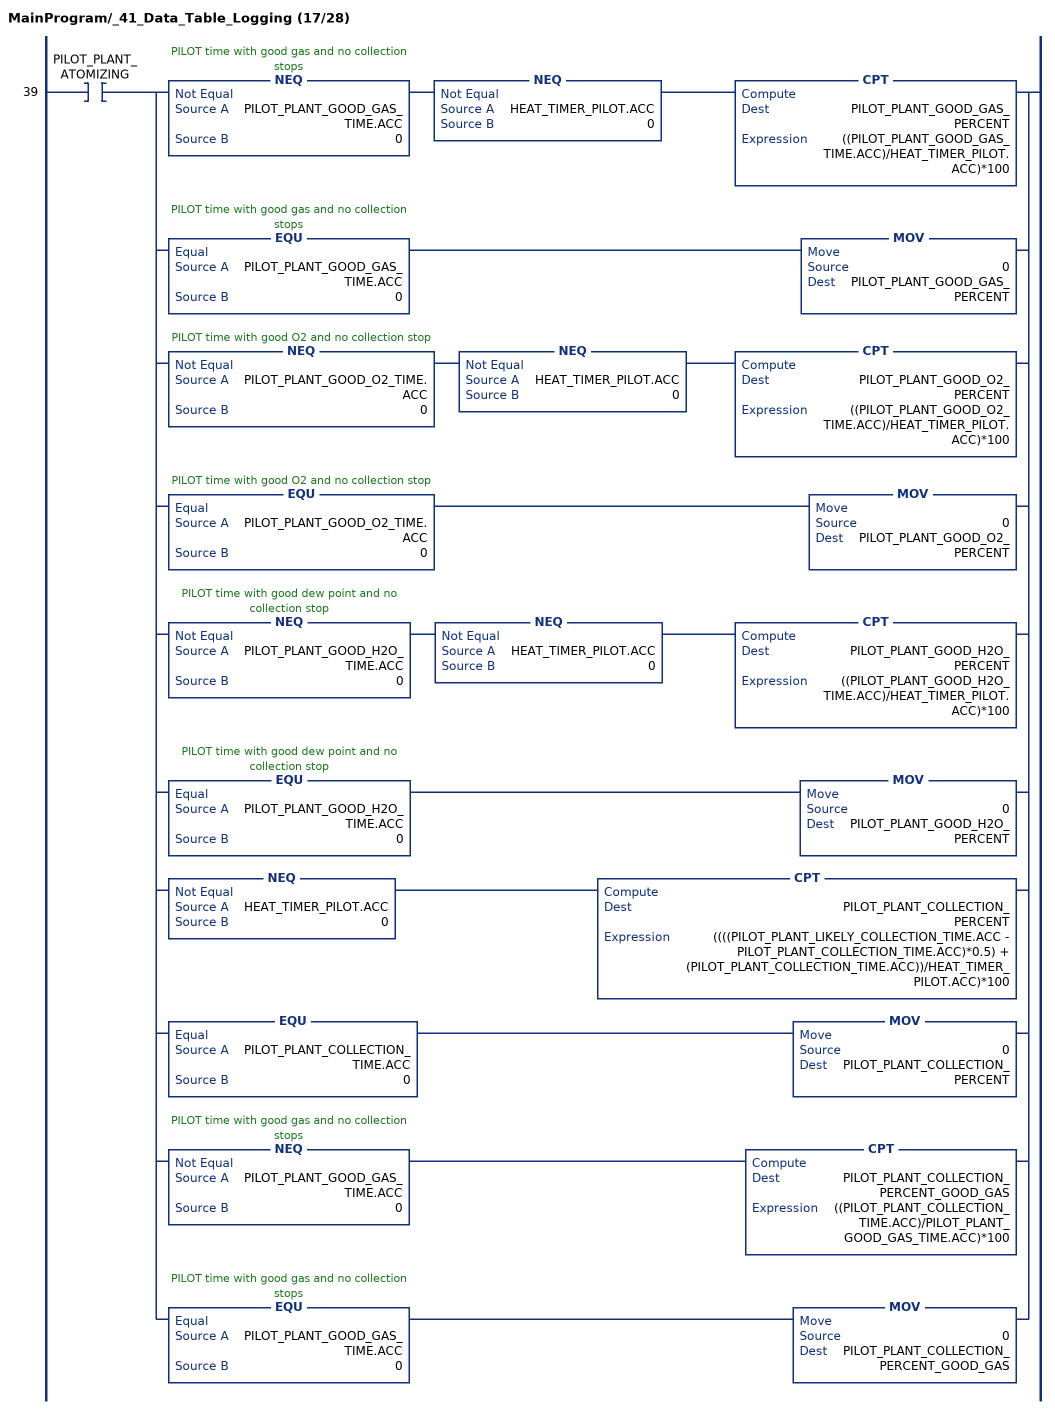
   39: XIC(PILOT_PLANT_ATOMIZING)[NEQ(PILOT_PLANT_GOOD_GAS_TIME.ACC,0) NEQ(HEAT_TIMER_PILOT.ACC,0) CPT(PILOT_PLANT_GOOD_GAS_PERCENT,((PILOT_PLANT_GOOD_GAS_TIME.ACC)/HEAT_TIMER_PILOT.ACC)*100) ,EQU(PILOT_PLANT_GOOD_GAS_TIME.ACC,0) MOV(0,PILOT_PLANT_GOOD_GAS_PERCENT) ,NEQ(PILOT_PLANT_GOOD_O2_TIME.ACC,0) NEQ(HEAT_TIMER_PILOT.ACC,0) CPT(PILOT_PLANT_GOOD_O2_PERCENT,((PILOT_PLANT_GOOD_O2_TIME.ACC)/HEAT_TIMER_PILOT.ACC)*100) ,EQU(PILOT_PLANT_GOOD_O2_TIME.ACC,0) MOV(0,PILOT_PLANT_GOOD_O2_PERCENT) ,NEQ(PILOT_PLANT_GOOD_H2O_TIME.ACC,0) NEQ(HEAT_TIMER_PILOT.ACC,0) CPT(PILOT_PLANT_GOOD_H2O_PERCENT,((PILOT_PLANT_GOOD_H2O_TIME.ACC)/HEAT_TIMER_PILOT.ACC)*100) ,EQU(PILOT_PLANT_GOOD_H2O_TIME.ACC,0) MOV(0,PILOT_PLANT_GOOD_H2O_PERCENT) ,NEQ(HEAT_TIMER_PILOT.ACC,0) CPT(PILOT_PLANT_COLLECTION_PERCENT,((((PILOT_PLANT_LIKELY_COLLECTION_TIME.ACC - PILOT_PLANT_COLLECTION_TIME.ACC)*0.5) + (PILOT_PLANT_COLLECTION_TIME.ACC))/HEAT_TIMER_PILOT.ACC)*100) ,EQU(PILOT_PLANT_COLLECTION_TIME.ACC,0) MOV(0,PILOT_PLANT_COLLECTION_PERCENT) ,NEQ(PILOT_PLANT_GOOD_GAS_TIME.ACC,0) CPT(PILOT_PLANT_COLLECTION_PERCENT_GOOD_GAS,((PILOT_PLANT_COLLECTION_TIME.ACC)/PILOT_PLANT_GOOD_GAS_TIME.ACC)*100) ,EQU(PILOT_PLANT_GOOD_GAS_TIME.ACC,0) MOV(0,PILOT_PLANT_COLLECTION_PERCENT_GOOD_GAS) ];
